(* CoDeSys 2.3.9.50 project: BallGame_template_with_PackMLandDriveFB.pro *)
(* Libraries: TcBase.lib 14.5.09 11:14:08, TcSystem.lib 7.6.16 10:01:22, STANDARD.LIB 5.6.98 11:03:02 *)

(* Task configuration *)
TASK BallGame (PRIORITY := 1, INTERVAL := T#10ms);
	PRG_HMI();
	MAIN();
END_TASK
TASK Drive (PRIORITY := 0, INTERVAL := T#5ms);
	PRG_Drive_Link();
END_TASK

(* Global variable list: Global_Variables *)
VAR_GLOBAL
(* -------------INPUTS and OUTPUTS -------------------*)
(* See Global_Variables_TwinCAT and Global_Variables_CodeSys for
environment specific physical IOs *)

(*-----------------------TIMERS----------------------------*)
	TONMove_Ball_Delay	: TON;
	TONDrive_Delay		: TON;

(*-----------------------COUNTERS----------------------------*)
	CountBallsSortedMetal			: INT:=0;	(*Balls sorted: Metal*)
	CountBallsSortedWooden		: INT:=0;	(*Balls sorted: Wood*)
	CountBallsSortedYellow		: INT:=0;	(*Balls sorted: Wood, Yellow*)
	CountBallsSortedRed			: INT:=0;	(*Balls sorted: Wood, Red*)
	CountBallsSortedBlue			: INT:=0;	(*Balls sorted: Wood, Blue*)
	CountBallsSortedGarbage		: INT:=0;	(*Balls sorted: Unknown*)
	arrCountBallsOnTubes	: ARRAY [1..4] OF INT;	(*Balls on tubes: 1=lower, 2=middle, 3=upper, 4=garbage*)

(*-----------------------FUNCTION BLOCKS----------------*)
	fbDrive				: FB_DriveMovement2;		(*FB for executing the motion*)
	fbStateModel			: FB_StateModel_ST;		(*FB for executing state model*)

(* -------------HMI INPUTS (from HMI to PLC) -------------------*)
	bHMI_BtnStart		: BOOL;		(*Start button on HMI*)
	HMI_uModeReq		: UINT :=1;

(* -------------HMI OUTPUTS (from PLC to HMI) -------------------*)
	PLC_uModeCurrent	: UINT;		(*Current Mode*)
	PLC_uStateCurrent	: UINT;		(*Current State*)
	O_Light_BeaconRed	: BOOL;		(*Light beacon: Red*)

(*-----------------------OTHER GLOBAL VARS ----------------*)


END_VAR

VAR_GLOBAL CONSTANT
(*-----------------------Lift Position Constants----------------------------*)
	GPOS_LOADING		: WORD := 16#0A;	(*Drive to loading level*)
	GPOS_PIPE_LOW	: WORD := 16#0B;	(*Drive to lower pipe*)
	GPOS_PIPE_MID		: WORD := 16#0C;	(*Drive to middle pipe*)
	GPOS_PIPE_UP		: WORD := 16#0D;	(*Drive to upper pipe*)
	GPOS_GARBAGE		: WORD := 16#0E;	(*Drive to garbage pipe*)
	GPOS_COLOR_SEN	: WORD := 16#0F;	(*Drive to colour sensor*)

(*-----------------------Ball Type Constants----------------------------*)
	METAL				: BOOL := FALSE;
	WOODEN		: BOOL := TRUE;

(*-----------------------TIME Constants----------------------------*)
	T_LOADING_BALL	: TIME := T#1.5s;	(*Delay for ball to roll from Slot2 to Lifter*)
	T_DRIVE_DELAY		: TIME := T#2s;	(*Delay for drive to start movement*)
END_VAR

(* Global variable list: Global_Variables_CodeSys *)
VAR_GLOBAL
(* -------------INPUTS-------------------*)
	ISensorOpt 			:BOOL;	(*Optical sensor - is ball present*)
	ISensorInd 			:BOOL;	(*Inductive sensor - is metal ball present*)
	IEmergencyClear 		:BOOL;	(*Emergency stop is cleared*)
	IRun 				:BOOL;	(*Run switch*)
	ILimitUp 				:BOOL;	(*Lift's limit switch is activated - Up*)
	ILimitLow 		 	:BOOL;	(*Lift's limit switch is activated - Low*)
	IGateClosedMid		:BOOL;	(*Pipe gate closed - Mid*)
	IGateClosedLow		:BOOL;	(*Pipe gate closed - Low*)
	ISorterGateClosed		:BOOL;	(*Sorter gate closed*)
	ISorterLiftUp			:BOOL;	(*Sorter lift at up position*)
	ISorterLiftDown		:BOOL;	(*Sorter lift at down position*)
	IPressureApplied		:BOOL;	(*Pressure is available for the system*)
	TEMP1				:BOOL;
	ISenColourYellow		:BOOL;	(*Colour sensor In1 - Yellow*)
	ISenColourBlue		:BOOL;	(*Colour sensor In2 - Blue*)
	ISenColourGreen		:BOOL;	(*Colour sensor In3 - Green*)
	ISenColourRed		:BOOL;	(*Colour sensor In4 - Red*)
	IDriveStatus 			:WORD;	(*From lift drive status information*)

(* -------------OUTPUTS-------------------*)
	OGateMid			:BOOL;	(*Valve: Open pipe gate - Mid*)
	OGateLow			:BOOL;	(*Valve: Open pipe gate - Low*)
	OSorterGate			:BOOL;	(*Valve: Open sorter gate*)
	OSorterLift			:BOOL;	(*Valve: Sorter lift up*)
	OEjector			:BOOL;	(*Ejector push ball out from lift*)
	ODriveControl 		:WORD;	(*To lift drive control information*)
END_VAR

(* Global variable list: Global_Variables_TwinCAT *)
VAR_GLOBAL
(* -------------INPUTS-------------------*)
	ISensorOpt 			AT %I*	:BOOL;	(*Optical sensor - is ball present*)
	ISensorInd 			AT %I*	:BOOL;	(*Inductive sensor - is metal ball present*)
	IEmergencyClear 	AT %I*	:BOOL;	(*Emergency stop is cleared*)
	IRun 				AT %I*	:BOOL;	(*Run switch*)
	ILimitUp 			AT %I*	:BOOL;	(*Lift's limit switch is activated - Up*)
	ILimitLow 			AT %I* 	:BOOL;	(*Lift's limit switch is activated - Low*)
	IGateClosedUp		AT %I* 	:BOOL;
	IGateClosedMid		AT %I*	:BOOL;	(*Pipe gate closed - Mid*)
	IGateClosedLow		AT %I*	:BOOL;	(*Pipe gate closed - Low*)
	ISorterGateClosed	AT %I*	:BOOL;	(*Sorter gate closed*)
	ISorterLiftUp		AT %I*	:BOOL;	(*Sorter lift at up position*)
	ISorterLiftDown		AT %I*	:BOOL;	(*Sorter lift at down position*)
	IPressureApplied	AT %I*	:BOOL;	(*Pressure is available for the system*)
	TEMP1				AT %I*	:BOOL;
	ISenColourYellow	AT %I*	:BOOL;	(*Colour sensor In1 - Yellow*)
	ISenColourBlue		AT %I*	:BOOL;	(*Colour sensor In2 - Blue*)
	ISenColourGreen		AT %I*	:BOOL;	(*Colour sensor In3 - Green*)
	ISenColourRed		AT %I*	:BOOL;	(*Colour sensor In4 - Red*)
	IDriveStatus 		AT %I*	:WORD;	(*From lift drive status information*)

(* -------------OUTPUTS-------------------*)
	OGateUp				AT %Q*	:BOOL;
	OGateMid			AT %Q*	:BOOL;	(*Valve: Open pipe gate - Mid*)
	OGateLow			AT %Q*	:BOOL;	(*Valve: Open pipe gate - Low*)
	OSorterGate			AT %Q*	:BOOL;	(*Valve: Open sorter gate*)
	OSorterLift			AT %Q*	:BOOL;	(*Valve: Sorter lift up*)
	OEjector			AT %Q*	:BOOL;	(*Ejector push ball out from lift*)
	ODriveControl 		AT %Q*	:WORD;	(*To lift drive control information*)

(* -------------HMI-------------------*)
	I_Btn_Reset		: BOOL;	(*Button: Reset*)
	I_Btn_Start		: BOOL;	(*Button: Start*)
	I_Btn_Stop		: BOOL;	(*Button: Stop*)
	I_Btn_EStop		: BOOL;	(*Button: Reset*)

(* -------------Drive-------------------*)
	bDriveEnabled 	: BOOL;

END_VAR

(* Global variable list: TwinCAT_Configuration *)
(* Generated automatically by TwinCAT - (read only) *)
VAR_CONFIG
	.ISensorOpt AT %IX0.0 : BOOL;	(*  ~ {LinkedWith:TIID^Device 4 (EL6731)^Box 2  (BK3110)^Term 2 (KL1002)^Channel 1^Input} *)
	.ISensorInd AT %IX0.1 : BOOL;	(*  ~ {LinkedWith:TIID^Device 4 (EL6731)^Box 2  (BK3110)^Term 2 (KL1002)^Channel 2^Input} *)
	.IEmergencyClear AT %IX0.2 : BOOL;	(*  ~ {LinkedWith:TIID^Device 4 (EL6731)^Box 2  (BK3110)^Term 3 (KL1002)^Channel 1^Input} *)
	.IRun AT %IX0.3 : BOOL;	(*  ~ {LinkedWith:TIID^Device 4 (EL6731)^Box 2  (BK3110)^Term 3 (KL1002)^Channel 2^Input} *)
	.ILimitUp AT %IX0.4 : BOOL;	(*  ~ {LinkedWith:TIID^Device 4 (EL6731)^Box 2  (BK3110)^Term 4 (KL1002)^Channel 1^Input} *)
	.ILimitLow AT %IX0.5 : BOOL;	(*  ~ {LinkedWith:TIID^Device 4 (EL6731)^Box 2  (BK3110)^Term 4 (KL1002)^Channel 2^Input} *)
	.IGateClosedUp AT %IX8.0 : BOOL;
	.IGateClosedMid AT %IX0.7 : BOOL;	(*  ~ {LinkedWith:TIID^Device 4 (EL6731)^Box 2  (BK3110)^Term 5 (KL1104)^Channel 2^Input} *)
	.IGateClosedLow AT %IX1.0 : BOOL;	(*  ~ {LinkedWith:TIID^Device 4 (EL6731)^Box 2  (BK3110)^Term 5 (KL1104)^Channel 3^Input} *)
	.ISorterGateClosed AT %IX1.1 : BOOL;	(*  ~ {LinkedWith:TIID^Device 4 (EL6731)^Box 2  (BK3110)^Term 5 (KL1104)^Channel 4^Input} *)
	.ISorterLiftUp AT %IX1.2 : BOOL;	(*  ~ {LinkedWith:TIID^Device 4 (EL6731)^Box 2  (BK3110)^Term 6 (KL1104)^Channel 1^Input} *)
	.ISorterLiftDown AT %IX1.3 : BOOL;	(*  ~ {LinkedWith:TIID^Device 4 (EL6731)^Box 2  (BK3110)^Term 6 (KL1104)^Channel 2^Input} *)
	.IPressureApplied AT %IX1.4 : BOOL;	(*  ~ {LinkedWith:TIID^Device 4 (EL6731)^Box 2  (BK3110)^Term 6 (KL1104)^Channel 3^Input} *)
	.TEMP1 AT %IX1.5 : BOOL;	(*  ~ {LinkedWith:TIID^Device 4 (EL6731)^Box 2  (BK3110)^Term 6 (KL1104)^Channel 4^Input} *)
	.ISenColourYellow AT %IX1.6 : BOOL;	(*  ~ {LinkedWith:TIID^Device 4 (EL6731)^Box 2  (BK3110)^Term 7 (KL1104)^Channel 1^Input} *)
	.ISenColourBlue AT %IX1.7 : BOOL;	(*  ~ {LinkedWith:TIID^Device 4 (EL6731)^Box 2  (BK3110)^Term 7 (KL1104)^Channel 2^Input} *)
	.ISenColourGreen AT %IX2.0 : BOOL;	(*  ~ {LinkedWith:TIID^Device 4 (EL6731)^Box 2  (BK3110)^Term 7 (KL1104)^Channel 3^Input} *)
	.ISenColourRed AT %IX2.1 : BOOL;	(*  ~ {LinkedWith:TIID^Device 4 (EL6731)^Box 2  (BK3110)^Term 7 (KL1104)^Channel 4^Input} *)
	.IDriveStatus AT %IB4 : WORD;	(*  ~ {LinkedWith:TIID^Device 4 (EL6731)^Box 5 (DKC03)^DKC03 mit LSPM2^Inputs^DKC03 mit LSPM2_0_0} *)
	.OGateUp AT %QX4.0 : BOOL;
	.OGateMid AT %QX0.1 : BOOL;	(*  ~ {LinkedWith:TIID^Device 4 (EL6731)^Box 2  (BK3110)^Term 8 (KL2114)^Channel 2^Output} *)
	.OGateLow AT %QX0.2 : BOOL;	(*  ~ {LinkedWith:TIID^Device 4 (EL6731)^Box 2  (BK3110)^Term 8 (KL2114)^Channel 3^Output} *)
	.OSorterGate AT %QX0.3 : BOOL;	(*  ~ {LinkedWith:TIID^Device 4 (EL6731)^Box 2  (BK3110)^Term 8 (KL2114)^Channel 4^Output} *)
	.OSorterLift AT %QX0.4 : BOOL;	(*  ~ {LinkedWith:TIID^Device 4 (EL6731)^Box 2  (BK3110)^Term 9 (KL2114)^Channel 1^Output} *)
	.OEjector AT %QX0.5 : BOOL;	(*  ~ {LinkedWith:TIID^Device 4 (EL6731)^Box 2  (BK3110)^Term 9 (KL2114)^Channel 2^Output} *)
	.ODriveControl AT %QB2 : WORD;	(*  ~ {LinkedWith:TIID^Device 4 (EL6731)^Box 5 (DKC03)^DKC03 mit LSPM2^Outputs^DKC03 mit LSPM2_1_0} *)
END_VAR

(* Data type *)
TYPE E_BallColour :
(
	NoColour := 0,
	Yellow := 1,
	Blue := 2,
	Red := 3
);
END_TYPE

(* Data type *)
TYPE E_ModeCtrl :
(
	eMode_undefined := 0,
	eMode_Automatic :=1,
	eMode_XXX :=2,
	eMode_Manual :=99
);
END_TYPE

(* Data type *)
TYPE E_ModeProc :
(*Procedural control modes. Can be changed in any state*)
(
	eModeProc_undefined := 0,
	eModeProc_Automatic :=1,
	eModeProc_SemiAutomatic :=2,
	eModeProc_Manual :=3
);
END_TYPE

(* Data type *)
TYPE E_State :
(
	eSt_Aborting :=0,
	eSt_Aborted,
	eSt_Clearing,
	eSt_Stopped,
	eSt_Stopping,
	eSt_Resetting,
	eSt_Idle,
	eSt_Starting,
	eSt_Execute,
	eSt_Suspending,
	eSt_Suspended,
	eSt_Unsuspending,
	eSt_Holding,
	eSt_Held,
	eSt_UnHolding,
	eSt_Completing,
	eSt_Completed
);
END_TYPE

(* POU PRG_HMI, ST *)
PROGRAM PRG_HMI
VAR
	(*HMI Buttons*)
	bBtnResetCounters	: BOOL;	(*Button Reset counters*)
	bBtnEmptyPipes		: BOOL;	(*Button Empty Pipes*)

	(*Variables for Lift visualisation*)
	iSorterLiftPos	: INT;		(*Position of Sorter Lift cylinder*)
	iLiftPos		: INT;		(*Position of the lift*)
	wTargetPos	: INT;		(*Current target position of the lift*)
	bBall_InLift	: BOOL;		(*Is there a ball in lift*)

	(*internal variables*)
	RS_Ball_InLift	: RS;		(*Flip-flop for ball in the lift*)
	i: INT := 0;		(*Counter*)
END_VAR
(*Producing blinking signal*)
PRG_Blinking();

(*Sorter lift position calculus*)
IF OSorterLift AND (iSorterLiftPos < 30) THEN
	iSorterLiftPos := iSorterLiftPos +1;
END_IF;
IF NOT OSorterLift AND (iSorterLiftPos > 0) THEN
	iSorterLiftPos := iSorterLiftPos - 1;
END_IF;

(*Lift position calculus*)
CASE fbDrive.wDestination OF
GPOS_PIPE_UP:		(*Go to Pipe Up*)
	wTargetPos:=375;
GPOS_PIPE_MID:	(*Go to Pipe Mid*)
	wTargetPos:=275;
GPOS_COLOR_SEN:	(*Go to Colour sensor*)
	wTargetPos:=220;
GPOS_PIPE_LOW:	(*Go to Pipe Low*)
	wTargetPos:=175;
GPOS_GARBAGE:	(*Go to garbage position*)
	wTargetPos:=110;
GPOS_LOADING:	(*Go to loading position*)
	wTargetPos:=20;
ELSE
	wTargetPos:=0;
END_CASE;

(*Drive lift*)
IF iLiftPos > wTargetPos THEN	(*Lift is higher than target*)
	iLiftPos := iLiftPos - 1;	 (*Go down*)
ELSIF iLiftPos < wTargetPos THEN	(*Lift is lower than target*)
	iLiftPos := iLiftPos + 1;	 (*Go up*)
END_IF;

(*Is there a ball in the lift*)
RS_Ball_InLift(
	SET:= (iLiftPos=20 AND NOT OSorterGate),
	RESET1:=OEjector ,
	Q1=>bBall_InLift );

(* ---------------------------------- Button handlers ---------------------------------- *)
(*Button Empty Pipes*)

(*Button Reset coutners*)
IF bBtnResetCounters THEN
	CountBallsSortedMetal := 0;
	CountBallsSortedWooden := 0;
	CountBallsSortedYellow := 0;
	CountBallsSortedBlue := 0;
	FOR i := 1 TO 3 DO
		arrCountBallsOnTubes[i] := 0;
	END_FOR;
END_IF;
END_PROGRAM

(* POU Programs/PRG_Blinking, ST *)
PROGRAM PRG_Blinking
(*Supporting caluculations: Blinking signals
Author: 	Niko Siltala, niko.siltala@tut.fi
Date: 	2014-01-01*)

VAR_OUTPUT
	bSign4Hz	:BOOL;				(*4 Hz (240krt/min) taajudella vaihteleva signaali*)
	bSign2Hz	:BOOL;				(*2 Hz (120krt/min) taajudella vaihteleva signaali*)
	bSign1Hz	:BOOL;				(*1 Hz (60krt/min) taajudella vaihteleva signaali*)
	bSign0_5Hz	:BOOL;				(*0,5 Hz (30krt/min) taajudella vaihteleva signaali*)
END_VAR
VAR
	bInitDone	: BOOL	:=FALSE;		(*Ohjelman initialisointi*)
	TP_Delay	: TP;					(*Nopein taajuus / 2 tuottaja*)
	bBaseHz	: BOOL	:=FALSE;		(*Nopein taajuus/2*)
	iBaseHz		: UINT	:=4;			(*Base taajuus (Hz)*)
	RTRIG_2Hz_Sign 	: R_TRIG;		(*2Hz signaalin generointi*)
	RTRIG_1Hz_Sign 	: R_TRIG;		(*1Hz signaalin generointi*)
	RTRIG_0_5Hz_Sign	: R_TRIG;	(*0,5Hz signaalin generointi*)
	tBaseTaajuus	:TIME;			(*Base vilkutuksen timerin arvo. f/2*)
	fPLC_CYCLE_TIME	: LREAL;		(*PLC:n cycli aika. Sekunttia*)
END_VAR
(*Ohjelman initialisoinnit - Suoritetaan vain kertaalleen*)
IF NOT bInitDone THEN
	fPLC_CYCLE_TIME := UDINT_TO_LREAL(SystemTaskInfoArr[1].cycleTime) / 10E6;
	(*Base Vilkkusignaalien tuottaminen*)
	(* 250ms - 1* cykliaika(20ms)*)
	tBaseTaajuus := LREAL_TO_TIME( ( (1/ UINT_TO_LREAL(iBaseHz) / 2 ) - 1 * fPLC_CYCLE_TIME ) * 1000);
	bInitDone := TRUE;
END_IF;


(*Base signaalin genrointi*)
TP_Delay(IN:=NOT TP_Delay.Q , PT:=tBaseTaajuus);
IF NOT TP_Delay.Q THEN
	bBaseHz := NOT bBaseHz;
	bSign4Hz:= bBaseHz;
END_IF;

(*2Hz signaalin genrointi*)
RTRIG_2Hz_Sign(CLK:=bSign4Hz);
IF RTRIG_2Hz_Sign.Q THEN
	bSign2Hz:=NOT bSign2Hz;
END_IF;

(*1Hz signaalin genrointi*)
RTRIG_1Hz_Sign(CLK:=bSign2Hz);
IF RTRIG_1Hz_Sign.Q THEN
	bSign1Hz:=NOT bSign1Hz;
END_IF;

(*0,5 Hz signaalin generointi*)
RTRIG_0_5Hz_Sign(CLK:=bSign1Hz);
IF (RTRIG_0_5Hz_Sign.Q) THEN
	bSign0_5Hz:= NOT bSign0_5Hz;
END_IF;
END_PROGRAM

(* POU MAIN, ST *)
PROGRAM MAIN
(*Main program for application. Uses PackML state model to control the execution of the application*)
VAR
	tonStarting			: TON;
	rsEmergencyClear	: RS;	(*RS - flip-flop for Emergency clear info*)
END_VAR
(* ****** Section 1: Initialisations and default values. Initial conditions for variables on every PLC cycle*)
(*Default values*)
fbStateModel.bSC := FALSE;
(*System resets*)

(* ****** Section 2: Actions in your program without considering the Control Mode. I.e. actions are performed same way indenpendent on
current Control Mode selection.*)
(*Mode independent state actions. Change / Add / Remove states according your need*)
CASE fbStateModel.eState OF
eSt_Aborting:
	(* One can make specific actions in case of specific Mode-State combination.
	   One can also consider to call a specific program when in specific Mode-State combination*)
	actAborting;
	fbStateModel.bSC := TRUE;		(*MODIFY*)
eSt_Clearing:
	fbStateModel.bSC := TRUE;		(*MODIFY*)
eSt_Resetting:
	fbStateModel.bSC := TRUE;
eSt_Holding:
	fbStateModel.bSC := TRUE;		(*MODIFY*)
eSt_UnHolding:
	fbStateModel.bSC := TRUE;		(*MODIFY*)
eSt_Suspending:
	fbStateModel.bSC := TRUE;		(*MODIFY*)
eSt_Unsuspending:
	fbStateModel.bSC := TRUE;		(*MODIFY*)
END_CASE;

(* ****** Section 3: Actions in your program which are Control Mode specific. Two nested case structures where outer one selects the
control mode and inner the PackML state. In order to avoid conflicts, it would be better to process each PackML state either in Section 2 
or Section 3, but not in both. *)
(*Execution mode related state actions. Change / Add / Remove mode and states according your need*)
CASE fbStateModel.eMode OF
(*MODE: MANUAL*)
eMode_Manual:
	(* ****** Section 3.1: PackML state based processing actions when Control Mode is Manual.*)
	CASE fbStateModel.eState OF
	eSt_Starting:
		IF IPressureApplied THEN
			fbStateModel.bSC := TRUE;			(*MODIFY*)
		END_IF
	eSt_Stopping:
		fbStateModel.bSC := TRUE;			(*MODIFY*)
	END_CASE;

(*MODE: AUTOMATIC*)
eMode_Automatic:
	(* ****** Section 3.2: PackML state based processing actions when Control Mode is Automatic.*)
	CASE fbStateModel.eState OF
	eSt_Idle:
		tonStarting(IN:=FALSE , PT:= , Q=> , ET=> );	(*MODIFY*)
	eSt_Starting:
		(* tonStarting(IN:=TRUE , PT:=T#2s , Q=> , ET=> );
		fbStateModel.bSC := tonStarting.Q; *)
		IF IPressureApplied THEN
			bDriveEnabled := TRUE;
			PRG_Initialisation(bReset:= , bExecute:= TRUE , bDone=> );
		END_IF

		IF PRG_Initialisation.bDone THEN
			PRG_Initialisation(bReset:= , bExecute:= FALSE , bDone=> );
			fbStateModel.bSC := TRUE;
		END_IF
	eSt_Completing:
		fbStateModel.bSC := TRUE;					(*MODIFY*)
	eSt_Completed:
		;
	END_CASE;

(* ****** Section 4: Grouping PackML states for calling Programs or FB instances.
This is to avoid repetition inside above case structure in Section 3. With IF clause setting lower (and upper) state limits we can filter out the states when we want to call 
specific programs. The order of states is defined in Tab:Data types > E_PackMLState. eSt_Aborting is lowest and eSt_Completed is highest.
Here we filter calling programs, only when we are in higher states than Stopped. 
This can be pulled out as completely separated section, like in PackML_StateModel_v2-2.pro project. There is inside IF again CASE which process each Control Mode separately.*)
(*Execution part. Making calls for program if we are on states above Stopped*)
	(*If we are between specific states, make some action or program call*)
	IF  (fbStateModel.eState>eSt_Starting) AND (fbStateModel.eState<=eSt_Completing) THEN
		(*Make here the actions / calls Good place to start with is PRG_Sorting (PRG)*)
		PRG_AutoSort(bExecute:= TRUE , bReset:= , bDone=> , bStopOk=> );
	END_IF;

(*MODE: UNKNOWN*)
ELSE	(*Error*)
	; (*TODO*)
END_CASE;

(* ****** Section 5: Calling the fbStateModel instance.
Here the instance of state model is called and all triggering inputs are set, but bSC (State Completed), which you control in your programs. 
This is indication that your program has  finished certain stage.
- Pay attention where the instance fbStateModel is defined. Do you do it in global variables or e.g. here in PRG_MAIN? Important is to use the 
same instance in all places, so that machine state is unique and shared. Remember, if you have multiple definitions, the PRG_MAIN "hides" 
the global one, and might lead to problems elswhere, when you think you are using the same instance, but actually are not. 
- In case you are using the PackML visualisation (VC_PackMLStates), make sure you connect its placeholder to the very same PackML FB instance.
- The Mask for wIgnoreState is created as following. I use binary base for the value(2#). The lowest bit in the mask corresponds the eSt_Aborting
 in E_PackMLState. The next is eSt_Aborted, and so on. Specific state is ignored and jumped over when it is masked out i.e. ignored by having 1 
in that position. Note that implementation allows this only for selected states. See FB_PackMLStateModel_ST code for further details.*)
(*Calling & Updating the state model*)
(*TODO: Evaluate and change all input conditions according your application needs*)
fbStateModel(
	bResetFB:= ,
	eModeReq:= HMI_uModeReq,
	wIgnoreState := 2#000000,		(*TODO: Which states should be ignodered. Default: 2#000000 or 2#100000. The latter is ignoring Resetting state*)
	bSC:= ,			(*Must not be assigned ANY variable, because fb input is directly operated!!!*)
	bAbort:= NOT (IEmergencyClear  OR  IPressureApplied),
	bClear:= IEmergencyClear,
	bReset:= I_Btn_Start,
	bStart:= I_Btn_Start,
	bHold:= ,
	bUn_Hold:= ,
	bSuspend:= ,
	bUn_Suspend:= ,
	bStop:= I_Btn_Stop ,
	bComplete:= ,
	bAck_Completed:= ,
	eMode=> PLC_uModeCurrent,
	eState=> PLC_uStateCurrent);

(* ****** Section 6: Here we update all outputs according the current state of our PackML model. This allows us to process the in single location.
The control of outputs is bind to state, not e.g. to inputs. The inputs are the one driving the PackML model forward. Again CASE structure can be used.*)
(*Call for HMI and UI update*)
(*PRG_Drive_Link()*);
HMI_and_UI_Update;
END_PROGRAM
ACTION actAborting:
bDriveEnabled := FALSE;
PRG_Sorting(bReset:=TRUE , bExecute:= FALSE);
END_ACTION
ACTION HMI_and_UI_Update:
(*Simulate emergency stop circuitry
rsEmergencyClear(
	SET:= I_Btn_Reset,
	RESET1:= I_Btn_EStop ,
	Q1=> IEmergencyClear);
*)

(*HMI Update*)
PRG_Blinking (bSign4Hz=> , bSign2Hz=> , bSign1Hz=> , bSign0_5Hz=> );
(*Init values*)
O_Light_BeaconRed := FALSE;

(*OLight_Start :=  (fbStateModel.eState >= eSt_Resetting) AND (fbStateModel.eState < eSt_Completed);*)
CASE fbStateModel.eState OF
eSt_Aborting, eSt_Aborted:
	O_Light_BeaconRed := PRG_Blinking.bSign1Hz;
eSt_Clearing:
	O_Light_BeaconRed := PRG_Blinking.bSign0_5Hz;
eSt_Stopped, eSt_Completed:
	O_Light_BeaconRed := TRUE;
eSt_Starting:
	;
END_CASE;
END_ACTION

(* POU Programs/PRG_Initialisation, SFC *)
PROGRAM PRG_Initialisation
(*Template program for system initialisation*)
VAR_INPUT
	bReset	: BOOL := FALSE;	(*Reseting the SFC*)
	bExecute	: BOOL;			(*Executes PRG*)
END_VAR
VAR_OUTPUT
	bDone		: BOOL;		(*Program operations done*)
END_VAR
VAR
(* -------------INTERNAL-------------------*)
	tonMoveDelay		: TON;
	tMoveDelay		: TIME := T#1s;
	bInitDone			: BOOL:=FALSE;	(*Initialisation done*)
	bGatesClosed	: BOOL:=FALSE;	(*Initialisation done*)
	bActuRetracted	: BOOL:=FALSE;
	bDriveAtLoading	: BOOL:=FALSE;

(*System variables. See SFC-flags: http://infosys.beckhoff.com/content/1033/tcplccontrol/html/tcplcctrl_editorsfc.htm?id=24319#SFC-Flags*)
	SFCReset		: BOOL := FALSE;	(*For reseting the SFC*)
END_VAR
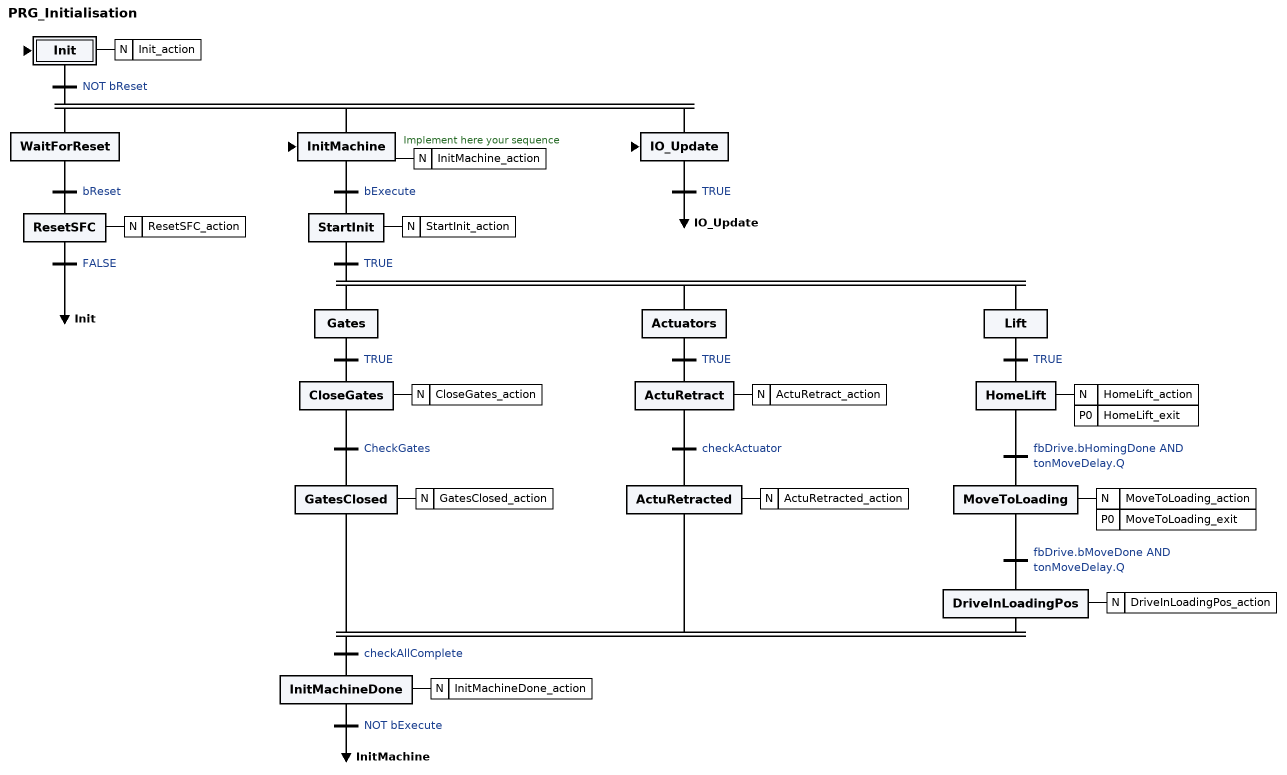
INITIAL_STEP Init:
	Init_action(N);
END_STEP
TRANSITION FROM Init TO (WaitForReset, InitMachine, IO_Update) := NOT bReset;
END_TRANSITION
STEP WaitForReset:
END_STEP
TRANSITION FROM WaitForReset TO ResetSFC := bReset;
END_TRANSITION
STEP InitMachine: (* Implement here your sequence *)
	InitMachine_action(N);
END_STEP
TRANSITION FROM InitMachine TO StartInit := bExecute;
END_TRANSITION
STEP StartInit:
	StartInit_action(N);
END_STEP
TRANSITION FROM StartInit TO (Gates, Actuators, Lift) := TRUE;
END_TRANSITION
STEP Gates:
END_STEP
TRANSITION FROM Gates TO CloseGates := TRUE;
END_TRANSITION
STEP CloseGates:
	CloseGates_action(N);
END_STEP
TRANSITION FROM CloseGates TO GatesClosed := CheckGates;
END_TRANSITION
STEP GatesClosed:
	GatesClosed_action(N);
END_STEP
STEP Actuators:
END_STEP
TRANSITION FROM Actuators TO ActuRetract := TRUE;
END_TRANSITION
STEP ActuRetract:
	ActuRetract_action(N);
END_STEP
TRANSITION FROM ActuRetract TO ActuRetracted := checkActuator;
END_TRANSITION
STEP ActuRetracted:
	ActuRetracted_action(N);
END_STEP
STEP Lift:
END_STEP
TRANSITION FROM Lift TO HomeLift := TRUE;
END_TRANSITION
STEP HomeLift:
	HomeLift_action(N);
	HomeLift_exit(P0);
END_STEP
TRANSITION FROM HomeLift TO MoveToLoading := fbDrive.bHomingDone AND tonMoveDelay.Q;
END_TRANSITION
STEP MoveToLoading:
	MoveToLoading_action(N);
	MoveToLoading_exit(P0);
END_STEP
TRANSITION FROM MoveToLoading TO DriveInLoadingPos := fbDrive.bMoveDone AND tonMoveDelay.Q;
END_TRANSITION
STEP DriveInLoadingPos:
	DriveInLoadingPos_action(N);
END_STEP
TRANSITION FROM (GatesClosed, ActuRetracted, DriveInLoadingPos) TO InitMachineDone := checkAllComplete;
END_TRANSITION
STEP InitMachineDone:
	InitMachineDone_action(N);
END_STEP
TRANSITION FROM InitMachineDone TO InitMachine := NOT bExecute;
END_TRANSITION
STEP IO_Update:
END_STEP
TRANSITION FROM IO_Update TO IO_Update := TRUE;
END_TRANSITION
STEP ResetSFC:
	ResetSFC_action(N);
END_STEP
TRANSITION FROM ResetSFC TO Init := FALSE;
END_TRANSITION

ACTION Init_action:
(*Clear Reset SFC*)
SFCReset:= FALSE;
bDone := FALSE;
END_ACTION

ACTION InitMachine_action:
(*Do some actions...

Sulje kaikki portit ... JA tarkista Steppiä seuraavassa transitioehdossa, että kaikki portit ovat kiinni
Close all gates.... and check in following transition that ALL gates are closed*)

;
END_ACTION

ACTION StartInit_action:
bDone := FALSE;
END_ACTION

ACTION CloseGates_action:
OGateUp		:= FALSE;
OGateMid	:= FALSE;
OGateLow	:= FALSE;
OSorterGate	:= FALSE;
END_ACTION

ACTION GatesClosed_action:
bGatesClosed := TRUE;
END_ACTION

ACTION ActuRetract_action:
OSorterLift	 := FALSE;
OEjector	 := FALSE;
END_ACTION

ACTION ActuRetracted_action:
bActuRetracted := TRUE;
END_ACTION

ACTION HomeLift_action:
fbDrive.bEnable := TRUE;
fbDrive.bStart := TRUE;
tonMoveDelay(IN:=TRUE , PT:= tMoveDelay);
END_ACTION

ACTION HomeLift_exit:
fbDrive.bStart:= FALSE;
tonMoveDelay(IN:=FALSE);
END_ACTION

ACTION MoveToLoading_action:
fbDrive.wTarget := GPOS_LOADING;
fbDrive.bStart:= TRUE;
tonMoveDelay(IN:=TRUE , PT:= tMoveDelay);
END_ACTION

ACTION MoveToLoading_exit:
fbDrive.bStart:= FALSE;
tonMoveDelay(IN:=FALSE);
END_ACTION

ACTION DriveInLoadingPos_action:
bDriveAtLoading := TRUE;
END_ACTION

ACTION InitMachineDone_action:
bDone := TRUE;
END_ACTION

ACTION ResetSFC_action:
(*Reset SFC*)
SFCReset:=TRUE;
END_ACTION

TRANSITION CheckGates:
_FBD_ (* Function Block Diagram *)
NETWORK 1
	AND(IGateClosedUp, IGateClosedMid, IGateClosedLow, ISorterGateClosed)
_END_FBD_
END_TRANSITION

TRANSITION checkActuator:
_FBD_ (* Function Block Diagram *)
NETWORK 1
	AND(ISorterLiftDown, NOT OEjector)
_END_FBD_
END_TRANSITION

TRANSITION checkAllComplete:
_FBD_ (* Function Block Diagram *)
NETWORK 1
	AND(bGatesClosed, bActuRetracted, bDriveAtLoading)
_END_FBD_
END_TRANSITION
END_PROGRAM

(* POU Programs/PRG_AutoSort, ST *)
PROGRAM PRG_AutoSort
VAR_INPUT
	bExecute	: BOOL;
	bReset	: BOOL := FALSE;
END_VAR
VAR_OUTPUT
	bDone		: BOOL;		(*Program operations done*)
	bStopOk    : BOOL;
END_VAR
VAR
	fbSorter	: FB_Sorter;
	fbLift		: FB_Lift;
	bBatchComplete  : BOOL := FALSE;
END_VAR
actUpdateIO;
actCheckAllOkStop;

CASE fbStateModel.eState OF
	eSt_Idle:
		fbStateModel.bComplete  := FALSE;
		fbStateModel.bSC 		:= TRUE;
	eSt_Resetting:
		fbStateModel.bSC := TRUE;
	eSt_Stopping:
		fbStateModel.bStop := FALSE;

		IF  bStopOk THEN
			fbStateModel.bSC := TRUE;
		END_IF
	eSt_Execute:
		fbSorter (bEnable :=  TRUE , bReset := FALSE);
		fbLift(bEnable :=  TRUE , bReset := FALSE);
		IF bBatchComplete  THEN
			fbStateModel.bComplete := TRUE;
		END_IF

	eSt_Completing:
		fbStateModel.bComplete := FALSE;
		IF bStopOK THEN
			fbStateModel.bSC := TRUE;
		END_IF

	eSt_Unsuspending:
		fbStateModel.bSC := TRUE;

	eSt_Suspending:
		fbStateModel.bSuspend := FALSE;
		fbStateModel.bSC := TRUE;

END_CASE
END_PROGRAM
ACTION actCheckAllOKStop:
IF fbSorter.bStopOK AND  fbLift.bStopOK THEN
	bStopOK := TRUE;
ELSE
	bStopOK := FALSE;
END_IF
END_ACTION
ACTION actUpdateIO:
fbSorter (
	bReset:= ,
	bEnable:= bExecute,
	I_SensorOpt:= ISensorOpt ,
	I_SensorInd:= ISensorInd,
	I_SorterLiftUp:= ISorterLiftUp ,
	I_SorterLiftDown:= ISorterLiftDown,
	hiRdyToReceive_FromDS:= fbLift.hoReadyToRecieve_ToUS ,
	hiBallAvail_FromUS:= ,
	bStopOK=> ,
	bBallLoaded=> ,
	bCurBallMetal=> ,
	O_SorterGate=> OSorterGate ,
	O_SorterLift=> OSorterLift ,
	hoBallAvail_ToDS=> ,
	hoReadyToRecieve_ToUS=> );

fbLift (
	bReset:= ,
	bEnable:= bExecute,
	I_LimitUp:= ILimitUp  ,
	I_LimitLow:= ILimitLow,
	I_WaitingBallMetal:= fbSorter.bCurBallMetal  ,
	I_SenColourYellow:= ISenColourYellow ,
	I_SenColourBlue:= ISenColourBlue ,
	I_SenColourGreen:= ISenColourGreen,
	I_SenColourRed:= ISenColourRed ,
	hiRdyToReceive_FromDS:= ,
	hiBallAvail_FromUS:= fbSorter.hoBallAvail_ToDS ,
	bStopOK=> ,
	bBallLoaded=> , 
	bCurBallMetal=> , 
	O_Ejector=> OEjector ,
	hoBallAvail_ToDS=> , 
	hoReadyToRecieve_ToUS=> );
END_ACTION

(* POU FBs/FB_Sorter, SFC *)
FUNCTION_BLOCK FB_Sorter
VAR_INPUT
	bReset			: BOOL;	(*Reset Request*)
	bEnable			: BOOL;
	I_SensorOpt		: BOOL;
	I_SensorInd		: BOOL;
	I_SorterLiftUp		: BOOL;
	I_SorterLiftDown	: BOOL;

	(*SMEMA Handshake Inputs*)
	hiRdyToReceive_FromDS	: BOOL;
	hiBallAvail_FromUS			: BOOL;
END_VAR
VAR_OUTPUT
	bStopOK			: BOOL;
	bBallLoaded		: BOOL;
	bCurBallMetal		: BOOL;
	O_SorterGate		: BOOL;
	O_SorterLift		: BOOL;

	(*SMEMA Handshake Outputs*)
	hoBallAvail_ToDS				: BOOL;
	hoReadyToRecieve_ToUS	: BOOL;
END_VAR
VAR
	tTransferDelay: TIME := T#2s;
	tMoveDelay	: TIME := T#1s;
	fbDelay		: FB_Wait;
	bLocalReset	: BOOL;	(*Performs local reset*)
	SFCReset 	: BOOL;	(*Resets the execution of SFC to init once this SFCFlag is set true *)
END_VAR
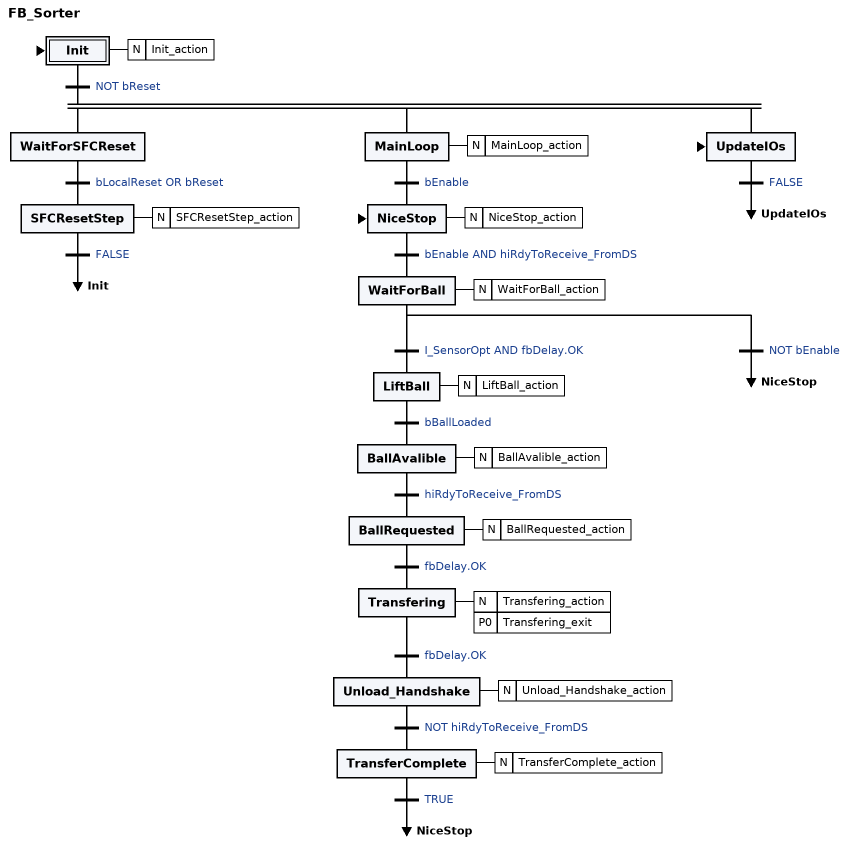
INITIAL_STEP Init:
	Init_action(N);
END_STEP
TRANSITION FROM Init TO (WaitForSFCReset, MainLoop, UpdateIOs) := NOT bReset;
END_TRANSITION
STEP WaitForSFCReset:
END_STEP
TRANSITION FROM WaitForSFCReset TO SFCResetStep := bLocalReset OR bReset;
END_TRANSITION
STEP MainLoop:
	MainLoop_action(N);
END_STEP
TRANSITION FROM MainLoop TO NiceStop := bEnable;
END_TRANSITION
STEP NiceStop:
	NiceStop_action(N);
END_STEP
TRANSITION FROM NiceStop TO WaitForBall := bEnable AND hiRdyToReceive_FromDS;
END_TRANSITION
STEP WaitForBall:
	WaitForBall_action(N);
END_STEP
TRANSITION FROM WaitForBall TO LiftBall := I_SensorOpt AND fbDelay.OK;
END_TRANSITION
TRANSITION FROM WaitForBall TO NiceStop := NOT bEnable;
END_TRANSITION
STEP LiftBall:
	LiftBall_action(N);
END_STEP
TRANSITION FROM LiftBall TO BallAvalible := bBallLoaded;
END_TRANSITION
STEP BallAvalible:
	BallAvalible_action(N);
END_STEP
TRANSITION FROM BallAvalible TO BallRequested := hiRdyToReceive_FromDS;
END_TRANSITION
STEP BallRequested:
	BallRequested_action(N);
END_STEP
TRANSITION FROM BallRequested TO Transfering := fbDelay.OK;
END_TRANSITION
STEP Transfering:
	Transfering_action(N);
	Transfering_exit(P0);
END_STEP
TRANSITION FROM Transfering TO Unload_Handshake := fbDelay.OK;
END_TRANSITION
STEP Unload_Handshake:
	Unload_Handshake_action(N);
END_STEP
TRANSITION FROM Unload_Handshake TO TransferComplete := NOT hiRdyToReceive_FromDS;
END_TRANSITION
STEP TransferComplete:
	TransferComplete_action(N);
END_STEP
TRANSITION FROM TransferComplete TO NiceStop := TRUE;
END_TRANSITION
STEP UpdateIOs:
END_STEP
TRANSITION FROM UpdateIOs TO UpdateIOs := FALSE;
END_TRANSITION
STEP SFCResetStep:
	SFCResetStep_action(N);
END_STEP
TRANSITION FROM SFCResetStep TO Init := FALSE;
END_TRANSITION

ACTION Init_action:
SFCReset := FALSE;
bLocalReset	:= FALSE;
bStopOK := FALSE;
END_ACTION

ACTION MainLoop_action:
hoBallAvail_ToDS			  := FALSE;
hoReadyToRecieve_ToUS := FALSE;
END_ACTION

ACTION NiceStop_action:
bBallLoaded 				  := FALSE;
bStopOK					  := TRUE;
hoBallAvail_ToDS			  := FALSE;
hoReadyToRecieve_ToUS := FALSE;
END_ACTION

ACTION WaitForBall_action:
fbDelay(IN_TIME:=tMoveDelay);
(* Move Lift Down *)
O_SorterLift := FALSE;
END_ACTION

ACTION LiftBall_action:
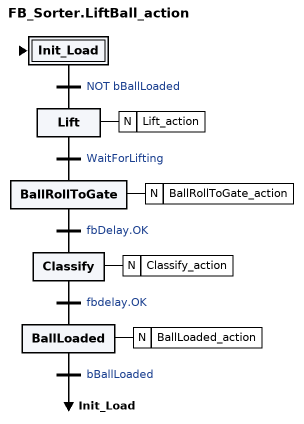
INITIAL_STEP Init_Load:
END_STEP
TRANSITION FROM Init_Load TO Lift := NOT bBallLoaded;
END_TRANSITION
STEP Lift:
	Lift_action(N);
END_STEP
TRANSITION FROM Lift TO BallRollToGate := WaitForLifting;
END_TRANSITION
STEP BallRollToGate:
	BallRollToGate_action(N);
END_STEP
TRANSITION FROM BallRollToGate TO Classify := fbDelay.OK;
END_TRANSITION
STEP Classify:
	Classify_action(N);
END_STEP
TRANSITION FROM Classify TO BallLoaded := fbdelay.OK;
END_TRANSITION
STEP BallLoaded:
	BallLoaded_action(N);
END_STEP
TRANSITION FROM BallLoaded TO Init_Load := bBallLoaded;
END_TRANSITION

ACTION Lift_action:
O_SorterLift := TRUE;
fbDelay(IN_TIME:=tMoveDelay);
END_ACTION

ACTION BallRollToGate_action:
fbDelay(IN_TIME:=tMoveDelay);
END_ACTION

ACTION Classify_action:
fbDelay(IN_TIME:=tMoveDelay);
IF I_SensorInd THEN
	bCurBallMetal := FALSE;
ELSE
	bCurBallMetal := TRUE;
END_IF
END_ACTION

ACTION BallLoaded_action:
bBallLoaded := TRUE;
END_ACTION

TRANSITION WaitForLifting:
_FBD_ (* Function Block Diagram *)
NETWORK 1
	AND(I_SorterLiftUp, fbDelay.OK)
_END_FBD_
END_TRANSITION
END_ACTION

ACTION BallAvalible_action:
hoBallAvail_ToDS := TRUE;
END_ACTION

ACTION BallRequested_action:
fbDelay(IN_TIME:=tMoveDelay);
END_ACTION

ACTION Transfering_action:
O_SorterGate := TRUE;
fbDelay(IN_TIME:=tTransferDelay);
END_ACTION

ACTION Transfering_exit:
O_SorterGate := FALSE;
END_ACTION

ACTION Unload_Handshake_action:
hoBallAvail_ToDS := FALSE;
END_ACTION

ACTION TransferComplete_action:
bBallLoaded := FALSE;
END_ACTION

ACTION SFCResetStep_action:
SFCReset := TRUE;
END_ACTION
END_FUNCTION_BLOCK

(* POU FBs/FB_Wait, ST *)
FUNCTION_BLOCK FB_Wait
(*Waits the given time and sets output after timer has run till end. When called again timer restarts.
Author: 	Niko Siltala, niko.siltala@tut.fi
Date: 	2014-01-01*)
VAR_INPUT
	IN_TIME	:TIME;		(*Time to wait*)
END_VAR
VAR_OUTPUT
	OK 		: BOOL:=FALSE;	(*Gets true after wait time has expired*)
END_VAR
VAR
	Timer	: TP;
	Falling	: F_TRIG;
END_VAR
IF Timer.Q=TRUE THEN
	(*Call timer block when pulse timer is counting*)
	Timer;
ELSE
	(*Timer has espired. Start it again*)
	Timer(IN:=FALSE);
	Timer(PT:=IN_TIME);
	Timer(IN:=TRUE);
END_IF;
(*Set output. True if timer has expired*)
OK:=NOT Timer.Q;
END_FUNCTION_BLOCK

(* POU FBs/FB_Lift, SFC *)
FUNCTION_BLOCK FB_Lift
VAR_INPUT
	bReset			 : BOOL;	(*Reset Request*)
	bEnable			 : BOOL;
	I_LimitUp 			 : BOOL;
	I_LimitLow 	        : BOOL;
	I_WaitingBallMetal : BOOL;

	(* ColourSensor *)
	I_SenColourYellow		:BOOL;	(*Colour sensor In1 - Yellow*)
	I_SenColourBlue		:BOOL;	(*Colour sensor In2 - Blue*)
	I_SenColourGreen		:BOOL;	(*Colour sensor In3 - Green*)
	I_SenColourRed		:BOOL;	(*Colour sensor In4 - Red*)

	(*SMEMA Handshake Inputs*)
	hiRdyToReceive_FromDS	: BOOL;
	hiBallAvail_FromUS			: BOOL;
END_VAR
VAR_OUTPUT
	bStopOK		: BOOL;
	bBallLoaded	: BOOL;
	bCurBallMetal	: BOOL;
	bCurrentBall 	: E_BallColour := NoColour;

	O_Ejector		:BOOL;

	(*SMEMA Handshake Outputs*)
	hoBallAvail_ToDS				: BOOL;
	hoReadyToRecieve_ToUS	: BOOL;
END_VAR
VAR
	bBallRequested : BOOL := FALSE;
	fbTransferBall	:FB_TransferBall2;

	fbDelay		: FB_Wait;
	tonMoveDelay	: TON;
	tonSensorDelay	: TON;
	tTransferDelay: TIME := T#4s;
	tMoveDelay	: TIME := T#4s;
	tSensorDelay	: TIME := T#2s;
	bLocalReset	: BOOL;	(*Performs local reset*)
	SFCReset 	: BOOL;	(*Resets the execution of SFC to init once this SFCFlag is set true *)
END_VAR
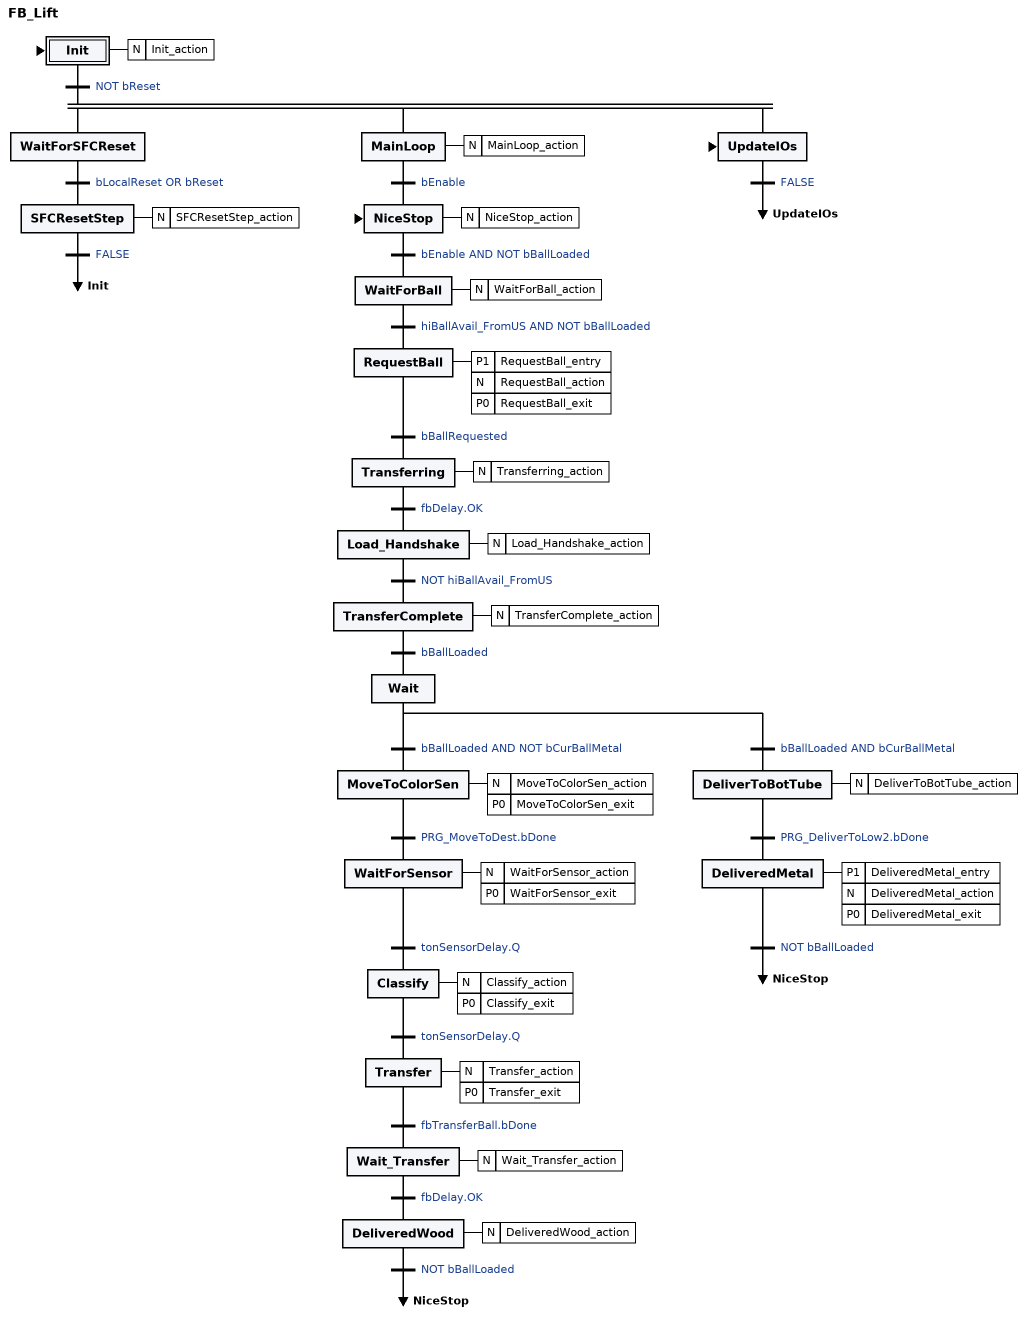
INITIAL_STEP Init:
	Init_action(N);
END_STEP
TRANSITION FROM Init TO (WaitForSFCReset, MainLoop, UpdateIOs) := NOT bReset;
END_TRANSITION
STEP WaitForSFCReset:
END_STEP
TRANSITION FROM WaitForSFCReset TO SFCResetStep := bLocalReset OR bReset;
END_TRANSITION
STEP MainLoop:
	MainLoop_action(N);
END_STEP
TRANSITION FROM MainLoop TO NiceStop := bEnable;
END_TRANSITION
STEP NiceStop:
	NiceStop_action(N);
END_STEP
TRANSITION FROM NiceStop TO WaitForBall := bEnable AND NOT bBallLoaded;
END_TRANSITION
STEP WaitForBall:
	WaitForBall_action(N);
END_STEP
TRANSITION FROM WaitForBall TO RequestBall := hiBallAvail_FromUS AND NOT bBallLoaded;
END_TRANSITION
STEP RequestBall:
	RequestBall_entry(P1);
	RequestBall_action(N);
	RequestBall_exit(P0);
END_STEP
TRANSITION FROM RequestBall TO Transferring := bBallRequested;
END_TRANSITION
STEP Transferring:
	Transferring_action(N);
END_STEP
TRANSITION FROM Transferring TO Load_Handshake := fbDelay.OK;
END_TRANSITION
STEP Load_Handshake:
	Load_Handshake_action(N);
END_STEP
TRANSITION FROM Load_Handshake TO TransferComplete := NOT hiBallAvail_FromUS;
END_TRANSITION
STEP TransferComplete:
	TransferComplete_action(N);
END_STEP
TRANSITION FROM TransferComplete TO Wait := bBallLoaded;
END_TRANSITION
STEP Wait:
END_STEP
TRANSITION FROM Wait TO MoveToColorSen := bBallLoaded AND NOT bCurBallMetal;
END_TRANSITION
TRANSITION FROM Wait TO DeliverToBotTube := bBallLoaded AND bCurBallMetal;
END_TRANSITION
STEP DeliverToBotTube:
	DeliverToBotTube_action(N);
END_STEP
TRANSITION FROM DeliverToBotTube TO DeliveredMetal := PRG_DeliverToLow2.bDone;
END_TRANSITION
STEP DeliveredMetal:
	DeliveredMetal_entry(P1);
	DeliveredMetal_action(N);
	DeliveredMetal_exit(P0);
END_STEP
TRANSITION FROM DeliveredMetal TO NiceStop := NOT bBallLoaded;
END_TRANSITION
STEP MoveToColorSen:
	MoveToColorSen_action(N);
	MoveToColorSen_exit(P0);
END_STEP
TRANSITION FROM MoveToColorSen TO WaitForSensor := PRG_MoveToDest.bDone;
END_TRANSITION
STEP WaitForSensor:
	WaitForSensor_action(N);
	WaitForSensor_exit(P0);
END_STEP
TRANSITION FROM WaitForSensor TO Classify := tonSensorDelay.Q;
END_TRANSITION
STEP Classify:
	Classify_action(N);
	Classify_exit(P0);
END_STEP
TRANSITION FROM Classify TO Transfer := tonSensorDelay.Q;
END_TRANSITION
STEP Transfer:
	Transfer_action(N);
	Transfer_exit(P0);
END_STEP
TRANSITION FROM Transfer TO Wait_Transfer := fbTransferBall.bDone;
END_TRANSITION
STEP Wait_Transfer:
	Wait_Transfer_action(N);
END_STEP
TRANSITION FROM Wait_Transfer TO DeliveredWood := fbDelay.OK;
END_TRANSITION
STEP DeliveredWood:
	DeliveredWood_action(N);
END_STEP
TRANSITION FROM DeliveredWood TO NiceStop := NOT bBallLoaded;
END_TRANSITION
STEP UpdateIOs:
END_STEP
TRANSITION FROM UpdateIOs TO UpdateIOs := FALSE;
END_TRANSITION
STEP SFCResetStep:
	SFCResetStep_action(N);
END_STEP
TRANSITION FROM SFCResetStep TO Init := FALSE;
END_TRANSITION

ACTION Init_action:
SFCReset := FALSE;
bLocalReset	:= FALSE;
END_ACTION

ACTION MainLoop_action:
hoBallAvail_ToDS			  := FALSE;
hoReadyToRecieve_ToUS := FALSE;
END_ACTION

ACTION NiceStop_action:
bStopOK	  	:= TRUE;
bCurrentBall	:= NoColour;
END_ACTION

ACTION WaitForBall_action:
bBallLoaded := FALSE;
hoReadyToRecieve_ToUS := TRUE;
END_ACTION

ACTION RequestBall_entry:
bStopOK := FALSE;
END_ACTION

ACTION RequestBall_action:
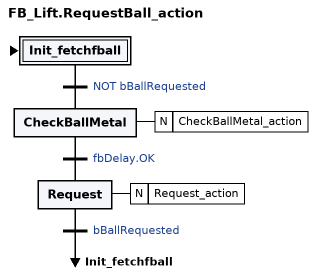
INITIAL_STEP Init_fetchfball:
END_STEP
TRANSITION FROM Init_fetchfball TO CheckBallMetal := NOT bBallRequested;
END_TRANSITION
STEP CheckBallMetal:
	CheckBallMetal_action(N);
END_STEP
TRANSITION FROM CheckBallMetal TO Request := fbDelay.OK;
END_TRANSITION
STEP Request:
	Request_action(N);
END_STEP
TRANSITION FROM Request TO Init_fetchfball := bBallRequested;
END_TRANSITION

ACTION CheckBallMetal_action:
bCurBallMetal	 := I_WaitingBallMetal;
fbDelay(IN_TIME:=T#2s);
END_ACTION

ACTION Request_action:
hoReadyToRecieve_ToUS := TRUE;
bBallRequested := TRUE;
END_ACTION
END_ACTION

ACTION RequestBall_exit:
bBallRequested := FALSE;
END_ACTION

ACTION Transferring_action:
fbDelay(IN_TIME:=tTransferDelay);
END_ACTION

ACTION Load_Handshake_action:
hoReadyToRecieve_ToUS := FALSE;
END_ACTION

ACTION TransferComplete_action:
bBallLoaded := TRUE;
END_ACTION

ACTION DeliverToBotTube_action:
PRG_DeliverToLow2(bExecute:=TRUE ,  bDone=> );
END_ACTION

ACTION DeliveredMetal_entry:
bBallLoaded := FALSE;
PRG_DeliverToLow(bReset:=FALSE , bExecute:=FALSE ,  bDone=> );
END_ACTION

ACTION DeliveredMetal_action:
bBallLoaded := FALSE;
END_ACTION

ACTION DeliveredMetal_exit:
PRG_DeliverToLow(bReset:=FALSE , bExecute:=FALSE ,  bDone=> );
END_ACTION

ACTION MoveToColorSen_action:
PRG_MoveToDest(bExecute:= TRUE, wTarget:= GPOS_COLOR_SEN, bDone:= );
END_ACTION

ACTION MoveToColorSen_exit:
PRG_MoveToDest( bExecute:=FALSE);
END_ACTION

ACTION WaitForSensor_action:
tonSensorDelay(IN:=TRUE , PT:= tSensorDelay);
END_ACTION

ACTION WaitForSensor_exit:
tonSensorDelay(IN:=FALSE);
END_ACTION

ACTION Classify_action:
tonSensorDelay(IN:=TRUE , PT:= tSensorDelay);
IF I_SenColourYellow THEN
	bCurrentBall := Yellow;
ELSIF  I_SenColourBlue THEN
	bCurrentBall := Blue;
ELSIF  I_SenColourRed THEN
	bCurrentBall := Red;
ELSE
	bCurrentBall := NoColour;
END_IF
END_ACTION

ACTION Classify_exit:
tonSensorDelay(IN:=FALSE);
END_ACTION

ACTION Transfer_action:
fbTransferBall(bExecute:= TRUE , bBallToTransfer:= bCurrentBall, bDone=> );
END_ACTION

ACTION Transfer_exit:
fbTransferBall(bExecute:= FALSE);
END_ACTION

ACTION Wait_Transfer_action:
fbDelay(IN_TIME:=tMoveDelay);
END_ACTION

ACTION DeliveredWood_action:
bBallLoaded := FALSE;
bCurrentBall := NoColour;
END_ACTION

ACTION SFCResetStep_action:
SFCReset := TRUE;
END_ACTION
END_FUNCTION_BLOCK

(* POU FBs/FB_TransferBall2, ST *)
FUNCTION_BLOCK FB_TransferBall2
VAR_INPUT
	bExecute			: BOOL;	(*enable and run*)
	bBallToTransfer 	: E_BallColour;
END_VAR
VAR_OUTPUT
	bDone			: BOOL;
	bActDone		: BOOL := FALSE;
END_VAR
VAR
	tonMoveDelay	: TON;
	tonEjectDelay	: TON;
	tMoveDelay	: TIME := T#1s;
	tEjectorDelay	: TIME := T#1s;
END_VAR
IF bExecute THEN
	CASE bBallToTransfer OF
		Yellow:
			PRG_MoveToDest(bExecute:= TRUE , wTarget:= GPOS_PIPE_UP, bDone:= );
			bDone	:= FALSE;
				(*IF PRG_MoveToDest.bDone THEN
					PRG_MoveToDest( bExecute:=FALSE);
					bDone	:= TRUE;
				END_IF*)
		Blue:
			PRG_MoveToDest(bExecute:= TRUE , wTarget:= GPOS_PIPE_MID, bDone:= );
				bDone	:= FALSE;
				(*IF PRG_MoveToDest.bDone THEN
					PRG_MoveToDest( bExecute:=FALSE);
					bDone	:= TRUE;
				END_IF*)
		Red, NoColour:
			PRG_MoveToDest(bExecute:= TRUE , wTarget:= GPOS_GARBAGE, bDone:= );
				bDone	:= FALSE;
				(*IF PRG_MoveToDest.bDone THEN
					PRG_MoveToDest( bExecute:=FALSE);
					bDone	:= TRUE;
				END_IF*)
	ELSE
		PRG_MoveToDest(bExecute:=FALSE);
		bDone	:= FALSE;
	END_CASE

	IF PRG_MoveToDest.bDone THEN
		PRG_MoveToDest(bExecute:=FALSE);
		bDone	:= TRUE;
	END_IF

ELSE
	bDone := FALSE;
END_IF
END_FUNCTION_BLOCK

(* POU Processes/PRG_MoveToDest, SFC *)
PROGRAM PRG_MoveToDest
VAR_INPUT
	bExecute: BOOL;
	wTarget : WORD;
END_VAR
VAR_INPUT
	bDone: BOOL;
END_VAR
VAR
	tonMoveDelay	: TON;
	tonEjectDelay	: TON;
	tonSensorDelay	: TON;
	tMoveDelay		: TIME := T#500ms;
	tEjectorDelay	: TIME := T#1s;
	tSensorDelay	: TIME := T#500ms;
END_VAR
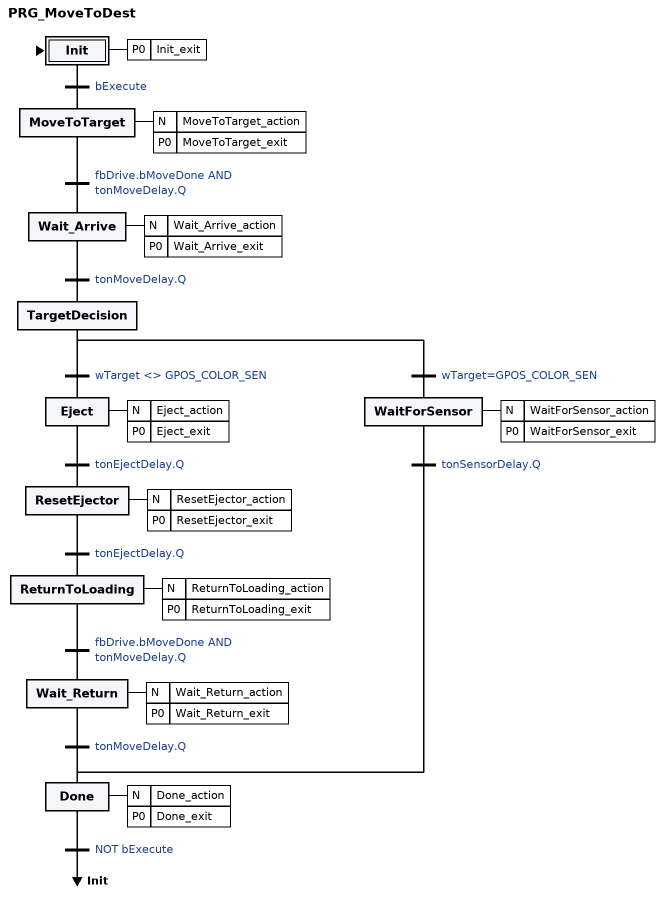
INITIAL_STEP Init:
	Init_exit(P0);
END_STEP
TRANSITION FROM Init TO MoveToTarget := bExecute;
END_TRANSITION
STEP MoveToTarget:
	MoveToTarget_action(N);
	MoveToTarget_exit(P0);
END_STEP
TRANSITION FROM MoveToTarget TO Wait_Arrive := fbDrive.bMoveDone AND tonMoveDelay.Q;
END_TRANSITION
STEP Wait_Arrive:
	Wait_Arrive_action(N);
	Wait_Arrive_exit(P0);
END_STEP
TRANSITION FROM Wait_Arrive TO TargetDecision := tonMoveDelay.Q;
END_TRANSITION
STEP TargetDecision:
END_STEP
TRANSITION FROM TargetDecision TO Eject := wTarget <> GPOS_COLOR_SEN;
END_TRANSITION
TRANSITION FROM TargetDecision TO WaitForSensor := wTarget=GPOS_COLOR_SEN;
END_TRANSITION
STEP WaitForSensor:
	WaitForSensor_action(N);
	WaitForSensor_exit(P0);
END_STEP
TRANSITION FROM WaitForSensor TO Done := tonSensorDelay.Q;
END_TRANSITION
STEP Eject:
	Eject_action(N);
	Eject_exit(P0);
END_STEP
TRANSITION FROM Eject TO ResetEjector := tonEjectDelay.Q;
END_TRANSITION
STEP ResetEjector:
	ResetEjector_action(N);
	ResetEjector_exit(P0);
END_STEP
TRANSITION FROM ResetEjector TO ReturnToLoading := tonEjectDelay.Q;
END_TRANSITION
STEP ReturnToLoading:
	ReturnToLoading_action(N);
	ReturnToLoading_exit(P0);
END_STEP
TRANSITION FROM ReturnToLoading TO Wait_Return := fbDrive.bMoveDone AND tonMoveDelay.Q;
END_TRANSITION
STEP Wait_Return:
	Wait_Return_action(N);
	Wait_Return_exit(P0);
END_STEP
TRANSITION FROM Wait_Return TO Done := tonMoveDelay.Q;
END_TRANSITION
STEP Done:
	Done_action(N);
	Done_exit(P0);
END_STEP
TRANSITION FROM Done TO Init := NOT bExecute;
END_TRANSITION

ACTION Init_exit:
bDone := FALSE;
END_ACTION

ACTION MoveToTarget_action:
tonMoveDelay(IN:=TRUE , PT:= tMoveDelay);
fbDrive(
	bEnable:= TRUE,
	bStart:= TRUE,
	wTarget:= wTarget);
END_ACTION

ACTION MoveToTarget_exit:
fbDrive(
	bStart:= FALSE);
tonMoveDelay(IN:=FALSE);
END_ACTION

ACTION Wait_Arrive_action:
tonMoveDelay(IN:=TRUE , PT:= tMoveDelay);
END_ACTION

ACTION Wait_Arrive_exit:
tonMoveDelay(IN:=FALSE);
END_ACTION

ACTION WaitForSensor_action:
tonSensorDelay(IN:=TRUE , PT:= tSensorDelay);
END_ACTION

ACTION WaitForSensor_exit:
tonSensorDelay(IN:=TRUE , PT:= tSensorDelay);
END_ACTION

ACTION Eject_action:
OEjector := TRUE;
tonEjectDelay(IN:=TRUE , PT:= tEjectorDelay);
END_ACTION

ACTION Eject_exit:
tonEjectDelay(IN:=FALSE);
END_ACTION

ACTION ResetEjector_action:
OEjector := FALSE;
tonEjectDelay(IN:=TRUE , PT:= tEjectorDelay);
END_ACTION

ACTION ResetEjector_exit:
tonEjectDelay(IN:=FALSE);
END_ACTION

ACTION ReturnToLoading_action:
fbDrive(
	bEnable:= TRUE,
	bStart:= TRUE,
	wTarget:= GPOS_LOADING);

tonMoveDelay(IN:=TRUE , PT:= tMoveDelay);
END_ACTION

ACTION ReturnToLoading_exit:
fbDrive(
	bStart:= FALSE);

tonMoveDelay(IN:=FALSE);
END_ACTION

ACTION Wait_Return_action:
tonMoveDelay(IN:=TRUE , PT:= tMoveDelay);
END_ACTION

ACTION Wait_Return_exit:
tonMoveDelay(IN:=FALSE);
END_ACTION

ACTION Done_action:
bDone := TRUE;
END_ACTION

ACTION Done_exit:
bDone := FALSE;
END_ACTION
END_PROGRAM

(* POU OLD/PRG_DeliverToLow2, SFC *)
PROGRAM PRG_DeliverToLow2
VAR_INPUT
	bExecute: BOOL;
END_VAR
VAR_INPUT
	bDone: BOOL;
END_VAR
VAR
	tonMoveDelay	: TON;
	tonEjectDelay	: TON;
	tMoveDelay	: TIME := T#4s;
	tEjectorDelay	: TIME := T#3s;
END_VAR
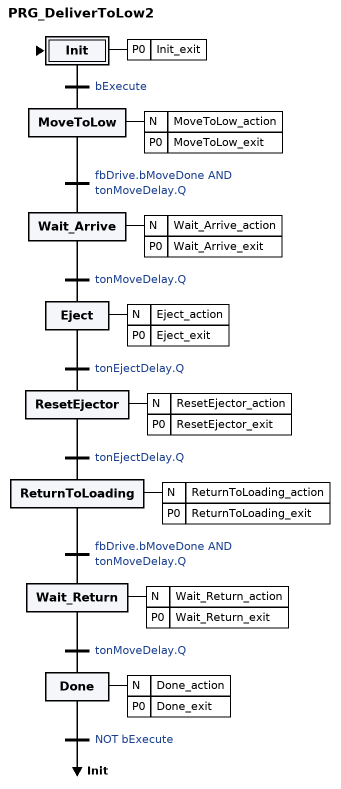
INITIAL_STEP Init:
	Init_exit(P0);
END_STEP
TRANSITION FROM Init TO MoveToLow := bExecute;
END_TRANSITION
STEP MoveToLow:
	MoveToLow_action(N);
	MoveToLow_exit(P0);
END_STEP
TRANSITION FROM MoveToLow TO Wait_Arrive := fbDrive.bMoveDone AND tonMoveDelay.Q;
END_TRANSITION
STEP Wait_Arrive:
	Wait_Arrive_action(N);
	Wait_Arrive_exit(P0);
END_STEP
TRANSITION FROM Wait_Arrive TO Eject := tonMoveDelay.Q;
END_TRANSITION
STEP Eject:
	Eject_action(N);
	Eject_exit(P0);
END_STEP
TRANSITION FROM Eject TO ResetEjector := tonEjectDelay.Q;
END_TRANSITION
STEP ResetEjector:
	ResetEjector_action(N);
	ResetEjector_exit(P0);
END_STEP
TRANSITION FROM ResetEjector TO ReturnToLoading := tonEjectDelay.Q;
END_TRANSITION
STEP ReturnToLoading:
	ReturnToLoading_action(N);
	ReturnToLoading_exit(P0);
END_STEP
TRANSITION FROM ReturnToLoading TO Wait_Return := fbDrive.bMoveDone AND tonMoveDelay.Q;
END_TRANSITION
STEP Wait_Return:
	Wait_Return_action(N);
	Wait_Return_exit(P0);
END_STEP
TRANSITION FROM Wait_Return TO Done := tonMoveDelay.Q;
END_TRANSITION
STEP Done:
	Done_action(N);
	Done_exit(P0);
END_STEP
TRANSITION FROM Done TO Init := NOT bExecute;
END_TRANSITION

ACTION Init_exit:
bDone := FALSE;
END_ACTION

ACTION MoveToLow_action:
tonMoveDelay(IN:=TRUE , PT:= tMoveDelay);
fbDrive(
	bEnable:= TRUE,
	bStart:= TRUE,
	wTarget:= GPOS_PIPE_LOW);
END_ACTION

ACTION MoveToLow_exit:
fbDrive(
	bStart:= FALSE);
tonMoveDelay(IN:=FALSE);
END_ACTION

ACTION Wait_Arrive_action:
tonMoveDelay(IN:=TRUE , PT:= tMoveDelay);
END_ACTION

ACTION Wait_Arrive_exit:
tonMoveDelay(IN:=FALSE);
END_ACTION

ACTION Eject_action:
OEjector := TRUE;
tonEjectDelay(IN:=TRUE , PT:= tEjectorDelay);
END_ACTION

ACTION Eject_exit:
tonEjectDelay(IN:=FALSE);
END_ACTION

ACTION ResetEjector_action:
OEjector := FALSE;
tonEjectDelay(IN:=TRUE , PT:= tEjectorDelay);
END_ACTION

ACTION ResetEjector_exit:
tonEjectDelay(IN:=FALSE);
END_ACTION

ACTION ReturnToLoading_action:
fbDrive(
	bEnable:= TRUE,
	bStart:= TRUE,
	wTarget:= GPOS_LOADING);

tonMoveDelay(IN:=TRUE , PT:= tMoveDelay);
END_ACTION

ACTION ReturnToLoading_exit:
fbDrive(
	bStart:= FALSE);

tonMoveDelay(IN:=FALSE);
END_ACTION

ACTION Wait_Return_action:
tonMoveDelay(IN:=TRUE , PT:= tMoveDelay);
END_ACTION

ACTION Wait_Return_exit:
tonMoveDelay(IN:=FALSE);
END_ACTION

ACTION Done_action:
bDone := TRUE;
END_ACTION

ACTION Done_exit:
bDone := FALSE;
END_ACTION
END_PROGRAM

(* POU OLD/PRG_DeliverToLow, SFC *)
PROGRAM PRG_DeliverToLow
VAR_INPUT
	bReset		: BOOL;	(*Reset program*)
	bExecute		: BOOL;	(*enable and run*)

END_VAR
VAR_OUTPUT
	bDone			: BOOL;
END_VAR
VAR
	tonMoveDelay	: TON;
	tonEjectDelay	: TON;
	SFCReset		: BOOL;

	tMoveDelay	: TIME := T#4s;
	tEjectorDelay	: TIME := T#3s;
END_VAR
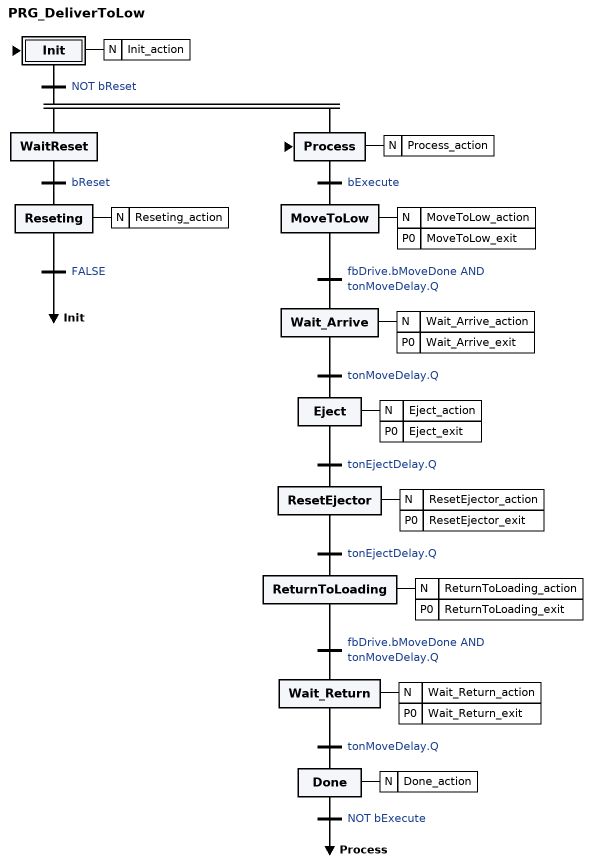
INITIAL_STEP Init:
	Init_action(N);
END_STEP
TRANSITION FROM Init TO (WaitReset, Process) := NOT bReset;
END_TRANSITION
STEP WaitReset:
END_STEP
TRANSITION FROM WaitReset TO Reseting := bReset;
END_TRANSITION
STEP Process:
	Process_action(N);
END_STEP
TRANSITION FROM Process TO MoveToLow := bExecute;
END_TRANSITION
STEP MoveToLow:
	MoveToLow_action(N);
	MoveToLow_exit(P0);
END_STEP
TRANSITION FROM MoveToLow TO Wait_Arrive := fbDrive.bMoveDone AND tonMoveDelay.Q;
END_TRANSITION
STEP Wait_Arrive:
	Wait_Arrive_action(N);
	Wait_Arrive_exit(P0);
END_STEP
TRANSITION FROM Wait_Arrive TO Eject := tonMoveDelay.Q;
END_TRANSITION
STEP Eject:
	Eject_action(N);
	Eject_exit(P0);
END_STEP
TRANSITION FROM Eject TO ResetEjector := tonEjectDelay.Q;
END_TRANSITION
STEP ResetEjector:
	ResetEjector_action(N);
	ResetEjector_exit(P0);
END_STEP
TRANSITION FROM ResetEjector TO ReturnToLoading := tonEjectDelay.Q;
END_TRANSITION
STEP ReturnToLoading:
	ReturnToLoading_action(N);
	ReturnToLoading_exit(P0);
END_STEP
TRANSITION FROM ReturnToLoading TO Wait_Return := fbDrive.bMoveDone AND tonMoveDelay.Q;
END_TRANSITION
STEP Wait_Return:
	Wait_Return_action(N);
	Wait_Return_exit(P0);
END_STEP
TRANSITION FROM Wait_Return TO Done := tonMoveDelay.Q;
END_TRANSITION
STEP Done:
	Done_action(N);
END_STEP
TRANSITION FROM Done TO Process := NOT bExecute;
END_TRANSITION
STEP Reseting:
	Reseting_action(N);
END_STEP
TRANSITION FROM Reseting TO Init := FALSE;
END_TRANSITION

ACTION Init_action:
SFCReset := FALSE;
bDone := FALSE;
END_ACTION

ACTION Process_action:
bDone := FALSE;
END_ACTION

ACTION MoveToLow_action:
bDone := FALSE;

fbDrive(
	bEnable:= TRUE,
	bStart:= TRUE,
	wTarget:= GPOS_PIPE_LOW);

tonMoveDelay(IN:=TRUE , PT:= tMoveDelay);
END_ACTION

ACTION MoveToLow_exit:
fbDrive(
	bStart:= FALSE);
tonMoveDelay(IN:=FALSE);
END_ACTION

ACTION Wait_Arrive_action:
tonMoveDelay(IN:=TRUE , PT:= tMoveDelay);
END_ACTION

ACTION Wait_Arrive_exit:
tonMoveDelay(IN:=FALSE);
END_ACTION

ACTION Eject_action:
OEjector := TRUE;
tonEjectDelay(IN:=TRUE , PT:= tEjectorDelay);
END_ACTION

ACTION Eject_exit:
tonEjectDelay(IN:=FALSE);
END_ACTION

ACTION ResetEjector_action:
OEjector := FALSE;
tonEjectDelay(IN:=TRUE , PT:= tEjectorDelay);
END_ACTION

ACTION ResetEjector_exit:
tonEjectDelay(IN:=FALSE);
END_ACTION

ACTION ReturnToLoading_action:
fbDrive(
	bEnable:= TRUE,
	bStart:= TRUE,
	wTarget:= GPOS_LOADING);

tonMoveDelay(IN:=TRUE , PT:= tMoveDelay);
END_ACTION

ACTION ReturnToLoading_exit:
fbDrive(
	bStart:= FALSE);

tonMoveDelay(IN:=FALSE);
END_ACTION

ACTION Wait_Return_action:
tonMoveDelay(IN:=TRUE , PT:= tMoveDelay);
END_ACTION

ACTION Wait_Return_exit:
tonMoveDelay(IN:=FALSE);
END_ACTION

ACTION Done_action:
bDone := TRUE;
END_ACTION

ACTION Reseting_action:
SFCReset := TRUE;
END_ACTION
END_PROGRAM

(* POU Programs/PRG_Drive_Link, FBD *)
PROGRAM PRG_Drive_Link
VAR
END_VAR
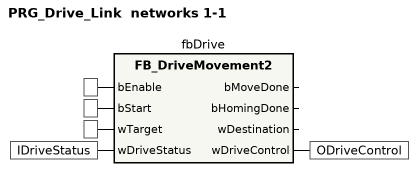
_FBD_ (* Function Block Diagram *)
NETWORK 1
	fbDrive:FB_DriveMovement2(bEnable: , bStart: , wTarget: , wDriveStatus: IDriveStatus, wDriveControl => ODriveControl)
_END_FBD_
END_PROGRAM

(* POU FBs/FB_DriveMovement2, ST *)
FUNCTION_BLOCK FB_DriveMovement2
(* This function block is making all movements for the drive
	bEnable = must be TRUE
	Target = int value of 0 - 63
	bStart = with rising edge starts the movement

	bMoveDone gets true when the movement is finalised.
Author: 	Niko Siltala, niko.siltala@tut.fi
Date: 	2014-01-01*)

VAR_INPUT
	bEnable			: BOOL:=FALSE;	(*Enables the fuction block*)
	bStart			: BOOL:=FALSE;	(*Starts the motion to target by rising edge*)
	wTarget			: WORD:=0;		(*Target destination*)
	wDriveStatus		: WORD;			(*Status word from Indramat Drive*)
END_VAR
VAR_OUTPUT
	bMoveDone		:BOOL:=FALSE;	(*The commanded move has been completed. Drive is at required destination*)
	bHomingDone	:BOOL:=FALSE;	(*Drive has been homed*)
	wDestination		:WORD;			(*Current destination*)
	wDriveControl		:WORD;			(*Control word to Indramat Drive*)
END_VAR
VAR_IN_OUT
END_VAR
VAR
	TONTimer1 	: TON;
	TONTimer2 	: TON;
END_VAR
(*
This function block is making all movements for the drive
	bEnable = must be TRUE
	Target = int value of 0 - 63
	bStart = with rising edge starts the movement

	bMoveDone gets true when the movement is finalised
*)
IF bEnable THEN
	(*Drive is Enabled*)
	wDriveControl:=wDriveControl OR 16#0001;
	IF (wDriveStatus AND 16#0080)>0 AND (wDriveStatus AND 16#0040)>0 THEN
		IF bStart=TRUE THEN
			(*bStart is true*)
			IF bHomingDone=FALSE THEN
				(*Homing procedure*)
				IF TONTimer1.Q=FALSE THEN
					wDriveControl:=16#0005;
					TONTimer1(IN:=TRUE, PT:=T#100ms);(*100ms*)
				ELSE
					IF TONTimer2.Q=FALSE THEN
						(*Start drive*)
						wDriveControl:=16#0007;
						TONTimer2(IN:=TRUE, PT:=T#500ms); (*500ms*)
					ELSE
						(*Timer2 have expired*)
						IF (wDriveStatus AND 16#0004)>0 THEN
							TONTimer1(IN:=FALSE);
							TONTimer2(IN:=FALSE);
							wDriveControl:=16#0001;
							bHomingDone:=TRUE;
						END_IF;
					END_IF;
				END_IF;
			ELSE
				(*Normal movement*)
				IF TONTimer1.Q=FALSE THEN
					(*Set target and Enabled*)
					wDriveControl:=SHL(wTarget,8) OR 16#0001;
					wDestination:=wTarget;
					TONTimer1(IN:=TRUE, PT:=T#10ms);(*10ms*)
				ELSE
					IF TONTimer2.Q=FALSE THEN
						(*Start drive*)
						wDriveControl:=wDriveControl OR 16#0002;
						TONTimer2(IN:=TRUE, PT:=T#500ms); (*500ms*)
					ELSE
						(*Timer2 have expired*)
						IF (wDriveStatus AND 16#0010)>0 THEN
							(*End the movement when user forgets to provide lowering edge*)
							(*bStart:=FALSE;*)
							(*Requested movement is done*)
							bMoveDone:=TRUE;
						END_IF;
					END_IF;
				END_IF; (*Normal movement*)
			END_IF;(*bHomingDone=FALSE*)
		ELSE
			(*bStart is false*)
			bMoveDone:=FALSE;
			TONTimer1(IN:=FALSE);
			TONTimer2(IN:=FALSE);
		END_IF;
	END_IF;
ELSE (*bEnable*)
	(*Drive is NOT Enabled*)
	wDriveControl:=16#0000;
	bMoveDone:=FALSE;
	bHomingDone:=FALSE;
	TONTimer1(IN:=FALSE);
	TONTimer2(IN:=FALSE);
END_IF;
END_FUNCTION_BLOCK

(* POU EXAMPLES, SFC *)
PROGRAM EXAMPLES
VAR
	fbDrive			: DriveMovement2;		(*FB for executing the motion*)
	tonTimer			: TON;			(*Standard TON timer. Use this*)
	fbDelay			: FB_Wait;		(*Different simplified timer.
END_VAR
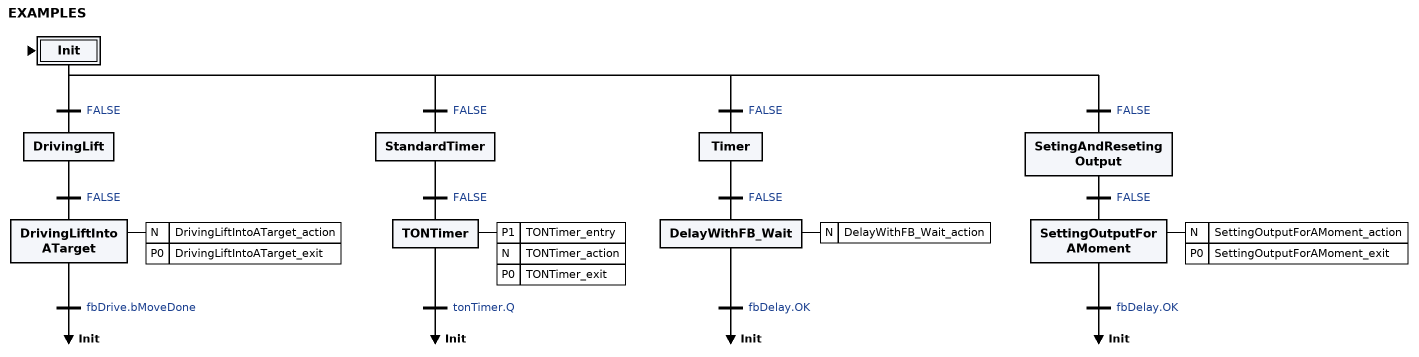
INITIAL_STEP Init:
END_STEP
TRANSITION FROM Init TO DrivingLift := FALSE;
END_TRANSITION
TRANSITION FROM Init TO StandardTimer := FALSE;
END_TRANSITION
TRANSITION FROM Init TO Timer := FALSE;
END_TRANSITION
TRANSITION FROM Init TO SetingAndResetingOutput := FALSE;
END_TRANSITION
STEP DrivingLift:
END_STEP
TRANSITION FROM DrivingLift TO DrivingLiftIntoATarget := FALSE;
END_TRANSITION
STEP DrivingLiftIntoATarget:
	DrivingLiftIntoATarget_action(N);
	DrivingLiftIntoATarget_exit(P0);
END_STEP
TRANSITION FROM DrivingLiftIntoATarget TO Init := fbDrive.bMoveDone;
END_TRANSITION
STEP StandardTimer:
END_STEP
TRANSITION FROM StandardTimer TO TONTimer := FALSE;
END_TRANSITION
STEP TONTimer:
	TONTimer_entry(P1);
	TONTimer_action(N);
	TONTimer_exit(P0);
END_STEP
TRANSITION FROM TONTimer TO Init := tonTimer.Q;
END_TRANSITION
STEP Timer:
END_STEP
TRANSITION FROM Timer TO DelayWithFB_Wait := FALSE;
END_TRANSITION
STEP DelayWithFB_Wait:
	DelayWithFB_Wait_action(N);
END_STEP
TRANSITION FROM DelayWithFB_Wait TO Init := fbDelay.OK;
END_TRANSITION
STEP SetingAndResetingOutput:
END_STEP
TRANSITION FROM SetingAndResetingOutput TO SettingOutputForAMoment := FALSE;
END_TRANSITION
STEP SettingOutputForAMoment:
	SettingOutputForAMoment_action(N);
	SettingOutputForAMoment_exit(P0);
END_STEP
TRANSITION FROM SettingOutputForAMoment TO Init := fbDelay.OK;
END_TRANSITION

ACTION DrivingLiftIntoATarget_action:
(*This executes and drives the lift to desired level (=wTarget)
wTarget is selected from given constants. See:Global Constants*)
fbDrive(
	bEnable:= TRUE,
	bStart:= TRUE,
	wTarget:= GPOS_LOADING);
END_ACTION

ACTION DrivingLiftIntoATarget_exit:
(*Stops the motion*)
fbDrive(
	bStart:= FALSE);
END_ACTION

ACTION TONTimer_entry:
tonTimer(IN:=FALSE);
END_ACTION

ACTION TONTimer_action:
tonTimer(IN:=TRUE , PT:=T#1s, Q=> , ET=> );
END_ACTION

ACTION TONTimer_exit:
tonTimer(IN:=FALSE);
END_ACTION

ACTION DelayWithFB_Wait_action:
(*Timer is counting*)
fbDelay(IN_TIME:=T#1s);
END_ACTION

ACTION SettingOutputForAMoment_action:
(*Timer is counting*)
fbDelay(IN_TIME:=T#500ms);

(*Setting Output*)
OEjector := TRUE;
END_ACTION

ACTION SettingOutputForAMoment_exit:
(*Clearing Output*)
OEjector := FALSE;
END_ACTION
END_PROGRAM

(* POU OLD/PRG_DeliverToGarbage, SFC *)
PROGRAM PRG_DeliverToGarbage
VAR_INPUT
	bReset		: BOOL;	(*Reset program*)
	bExecute		: BOOL;	(*enable and run*)
END_VAR
VAR_OUTPUT
	bDone			: BOOL;
END_VAR
VAR
	tonMoveDelay	: TON;
	tonEjectDelay	: TON;
	SFCReset		: BOOL;

	tMoveDelay	: TIME := T#4s;
	tEjectorDelay	: TIME := T#2s;
END_VAR
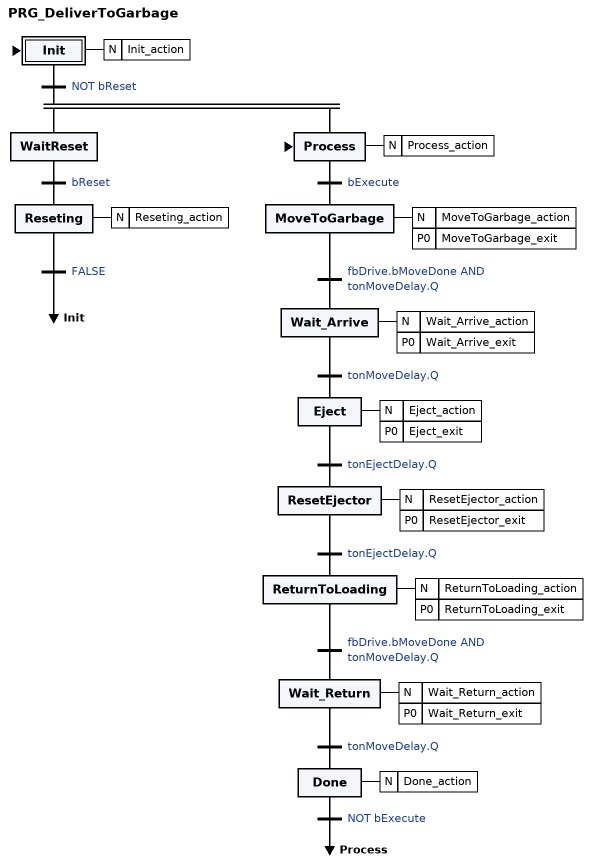
INITIAL_STEP Init:
	Init_action(N);
END_STEP
TRANSITION FROM Init TO (WaitReset, Process) := NOT bReset;
END_TRANSITION
STEP WaitReset:
END_STEP
TRANSITION FROM WaitReset TO Reseting := bReset;
END_TRANSITION
STEP Process:
	Process_action(N);
END_STEP
TRANSITION FROM Process TO MoveToGarbage := bExecute;
END_TRANSITION
STEP MoveToGarbage:
	MoveToGarbage_action(N);
	MoveToGarbage_exit(P0);
END_STEP
TRANSITION FROM MoveToGarbage TO Wait_Arrive := fbDrive.bMoveDone AND tonMoveDelay.Q;
END_TRANSITION
STEP Wait_Arrive:
	Wait_Arrive_action(N);
	Wait_Arrive_exit(P0);
END_STEP
TRANSITION FROM Wait_Arrive TO Eject := tonMoveDelay.Q;
END_TRANSITION
STEP Eject:
	Eject_action(N);
	Eject_exit(P0);
END_STEP
TRANSITION FROM Eject TO ResetEjector := tonEjectDelay.Q;
END_TRANSITION
STEP ResetEjector:
	ResetEjector_action(N);
	ResetEjector_exit(P0);
END_STEP
TRANSITION FROM ResetEjector TO ReturnToLoading := tonEjectDelay.Q;
END_TRANSITION
STEP ReturnToLoading:
	ReturnToLoading_action(N);
	ReturnToLoading_exit(P0);
END_STEP
TRANSITION FROM ReturnToLoading TO Wait_Return := fbDrive.bMoveDone AND tonMoveDelay.Q;
END_TRANSITION
STEP Wait_Return:
	Wait_Return_action(N);
	Wait_Return_exit(P0);
END_STEP
TRANSITION FROM Wait_Return TO Done := tonMoveDelay.Q;
END_TRANSITION
STEP Done:
	Done_action(N);
END_STEP
TRANSITION FROM Done TO Process := NOT bExecute;
END_TRANSITION
STEP Reseting:
	Reseting_action(N);
END_STEP
TRANSITION FROM Reseting TO Init := FALSE;
END_TRANSITION

ACTION Init_action:
SFCReset := FALSE;
bDone := FALSE;
END_ACTION

ACTION Process_action:
bDone := FALSE;
END_ACTION

ACTION MoveToGarbage_action:
bDone := FALSE;

fbDrive(
	bEnable:= TRUE,
	bStart:= TRUE,
	wTarget:= GPOS_GARBAGE);

tonMoveDelay(IN:=TRUE , PT:= tMoveDelay);
END_ACTION

ACTION MoveToGarbage_exit:
fbDrive(
	bStart:= FALSE);

tonMoveDelay(IN:=FALSE);
END_ACTION

ACTION Wait_Arrive_action:
tonMoveDelay(IN:=TRUE , PT:= tMoveDelay);
END_ACTION

ACTION Wait_Arrive_exit:
tonMoveDelay(IN:=FALSE);
END_ACTION

ACTION Eject_action:
OEjector := TRUE;
tonEjectDelay(IN:=TRUE , PT:= tEjectorDelay);
END_ACTION

ACTION Eject_exit:
tonEjectDelay(IN:=FALSE);
END_ACTION

ACTION ResetEjector_action:
OEjector := FALSE;
tonEjectDelay(IN:=TRUE , PT:= tEjectorDelay);
END_ACTION

ACTION ResetEjector_exit:
tonEjectDelay(IN:=FALSE);
END_ACTION

ACTION ReturnToLoading_action:
fbDrive(
	bEnable:= TRUE,
	bStart:= TRUE,
	wTarget:= GPOS_LOADING);

tonMoveDelay(IN:=TRUE , PT:= tMoveDelay);
END_ACTION

ACTION ReturnToLoading_exit:
fbDrive(
	bStart:= FALSE);

tonMoveDelay(IN:=FALSE);
END_ACTION

ACTION Wait_Return_action:
tonMoveDelay(IN:=TRUE , PT:= tMoveDelay);
END_ACTION

ACTION Wait_Return_exit:
tonMoveDelay(IN:=FALSE);
END_ACTION

ACTION Done_action:
bDone := TRUE;
END_ACTION

ACTION Reseting_action:
SFCReset := TRUE;
END_ACTION
END_PROGRAM

(* POU OLD/PRG_DeliverToGarbage2, SFC *)
PROGRAM PRG_DeliverToGarbage2
VAR_INPUT
	bExecute: BOOL;
END_VAR
VAR_INPUT
	bDone: BOOL;
END_VAR
VAR
	tonMoveDelay	: TON;
	tonEjectDelay	: TON;
	tMoveDelay	: TIME := T#3s;
	tEjectorDelay	: TIME := T#3s;
END_VAR
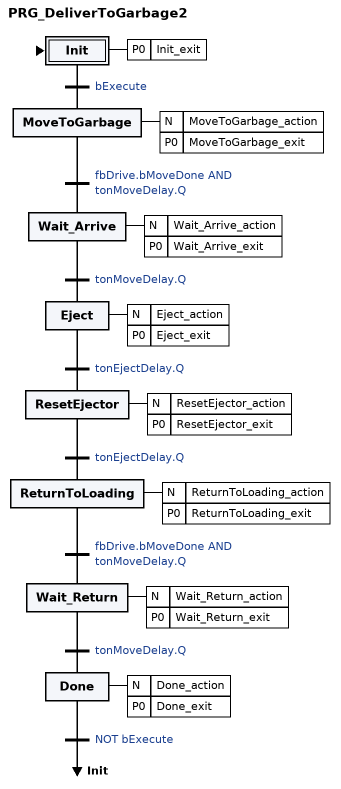
INITIAL_STEP Init:
	Init_exit(P0);
END_STEP
TRANSITION FROM Init TO MoveToGarbage := bExecute;
END_TRANSITION
STEP MoveToGarbage:
	MoveToGarbage_action(N);
	MoveToGarbage_exit(P0);
END_STEP
TRANSITION FROM MoveToGarbage TO Wait_Arrive := fbDrive.bMoveDone AND tonMoveDelay.Q;
END_TRANSITION
STEP Wait_Arrive:
	Wait_Arrive_action(N);
	Wait_Arrive_exit(P0);
END_STEP
TRANSITION FROM Wait_Arrive TO Eject := tonMoveDelay.Q;
END_TRANSITION
STEP Eject:
	Eject_action(N);
	Eject_exit(P0);
END_STEP
TRANSITION FROM Eject TO ResetEjector := tonEjectDelay.Q;
END_TRANSITION
STEP ResetEjector:
	ResetEjector_action(N);
	ResetEjector_exit(P0);
END_STEP
TRANSITION FROM ResetEjector TO ReturnToLoading := tonEjectDelay.Q;
END_TRANSITION
STEP ReturnToLoading:
	ReturnToLoading_action(N);
	ReturnToLoading_exit(P0);
END_STEP
TRANSITION FROM ReturnToLoading TO Wait_Return := fbDrive.bMoveDone AND tonMoveDelay.Q;
END_TRANSITION
STEP Wait_Return:
	Wait_Return_action(N);
	Wait_Return_exit(P0);
END_STEP
TRANSITION FROM Wait_Return TO Done := tonMoveDelay.Q;
END_TRANSITION
STEP Done:
	Done_action(N);
	Done_exit(P0);
END_STEP
TRANSITION FROM Done TO Init := NOT bExecute;
END_TRANSITION

ACTION Init_exit:
bDone := FALSE;
END_ACTION

ACTION MoveToGarbage_action:
fbDrive(
	bEnable:= TRUE,
	bStart:= TRUE,
	wTarget:= GPOS_GARBAGE);

tonMoveDelay(IN:=TRUE , PT:= tMoveDelay);
END_ACTION

ACTION MoveToGarbage_exit:
fbDrive(
	bStart:= FALSE);
tonMoveDelay(IN:=FALSE);
END_ACTION

ACTION Wait_Arrive_action:
tonMoveDelay(IN:=TRUE , PT:= tMoveDelay);
END_ACTION

ACTION Wait_Arrive_exit:
tonMoveDelay(IN:=FALSE);
END_ACTION

ACTION Eject_action:
OEjector := TRUE;
tonEjectDelay(IN:=TRUE , PT:= tEjectorDelay);
END_ACTION

ACTION Eject_exit:
tonEjectDelay(IN:=FALSE);
END_ACTION

ACTION ResetEjector_action:
OEjector := FALSE;
tonEjectDelay(IN:=TRUE , PT:= tEjectorDelay);
END_ACTION

ACTION ResetEjector_exit:
tonEjectDelay(IN:=FALSE);
END_ACTION

ACTION ReturnToLoading_action:
fbDrive(
	bEnable:= TRUE,
	bStart:= TRUE,
	wTarget:= GPOS_LOADING);

tonMoveDelay(IN:=TRUE , PT:= tMoveDelay);
END_ACTION

ACTION ReturnToLoading_exit:
fbDrive(
	bStart:= FALSE);

tonMoveDelay(IN:=FALSE);
END_ACTION

ACTION Wait_Return_action:
tonMoveDelay(IN:=TRUE , PT:= tMoveDelay);
END_ACTION

ACTION Wait_Return_exit:
tonMoveDelay(IN:=FALSE);
END_ACTION

ACTION Done_action:
bDone := TRUE;
END_ACTION

ACTION Done_exit:
bDone := FALSE;
END_ACTION
END_PROGRAM

(* POU OLD/PRG_DeliverToMid, SFC *)
PROGRAM PRG_DeliverToMid
VAR_INPUT
	bReset		: BOOL;	(*Reset program*)
	bExecute		: BOOL;	(*enable and run*)
END_VAR
VAR_OUTPUT
	bDone			: BOOL;
END_VAR
VAR
	tonMoveDelay	: TON;
	tonEjectDelay	: TON;
	SFCReset		: BOOL;

	tMoveDelay	: TIME := T#4s;
	tEjectorDelay	: TIME := T#2s;
END_VAR
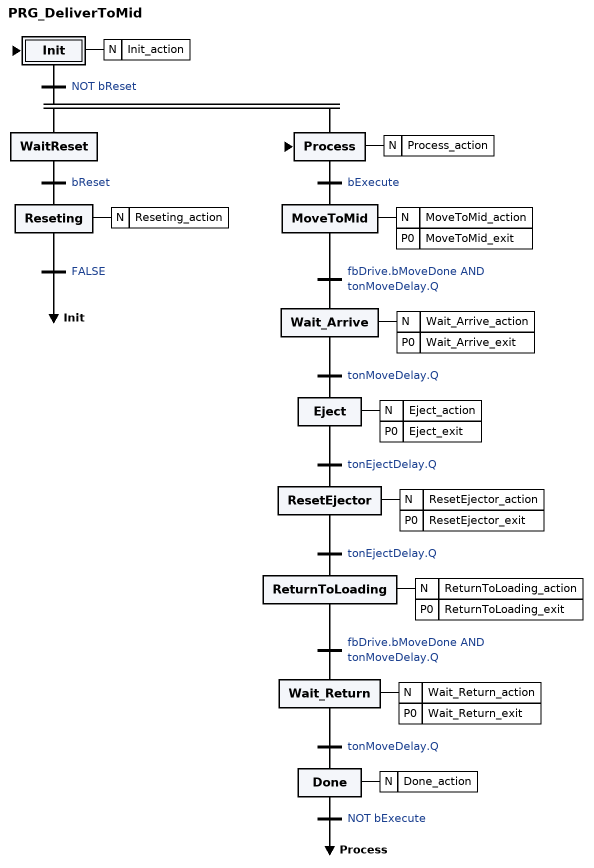
INITIAL_STEP Init:
	Init_action(N);
END_STEP
TRANSITION FROM Init TO (WaitReset, Process) := NOT bReset;
END_TRANSITION
STEP WaitReset:
END_STEP
TRANSITION FROM WaitReset TO Reseting := bReset;
END_TRANSITION
STEP Process:
	Process_action(N);
END_STEP
TRANSITION FROM Process TO MoveToMid := bExecute;
END_TRANSITION
STEP MoveToMid:
	MoveToMid_action(N);
	MoveToMid_exit(P0);
END_STEP
TRANSITION FROM MoveToMid TO Wait_Arrive := fbDrive.bMoveDone AND tonMoveDelay.Q;
END_TRANSITION
STEP Wait_Arrive:
	Wait_Arrive_action(N);
	Wait_Arrive_exit(P0);
END_STEP
TRANSITION FROM Wait_Arrive TO Eject := tonMoveDelay.Q;
END_TRANSITION
STEP Eject:
	Eject_action(N);
	Eject_exit(P0);
END_STEP
TRANSITION FROM Eject TO ResetEjector := tonEjectDelay.Q;
END_TRANSITION
STEP ResetEjector:
	ResetEjector_action(N);
	ResetEjector_exit(P0);
END_STEP
TRANSITION FROM ResetEjector TO ReturnToLoading := tonEjectDelay.Q;
END_TRANSITION
STEP ReturnToLoading:
	ReturnToLoading_action(N);
	ReturnToLoading_exit(P0);
END_STEP
TRANSITION FROM ReturnToLoading TO Wait_Return := fbDrive.bMoveDone AND tonMoveDelay.Q;
END_TRANSITION
STEP Wait_Return:
	Wait_Return_action(N);
	Wait_Return_exit(P0);
END_STEP
TRANSITION FROM Wait_Return TO Done := tonMoveDelay.Q;
END_TRANSITION
STEP Done:
	Done_action(N);
END_STEP
TRANSITION FROM Done TO Process := NOT bExecute;
END_TRANSITION
STEP Reseting:
	Reseting_action(N);
END_STEP
TRANSITION FROM Reseting TO Init := FALSE;
END_TRANSITION

ACTION Init_action:
SFCReset := FALSE;
bDone := FALSE;
END_ACTION

ACTION Process_action:
bDone := FALSE;
END_ACTION

ACTION MoveToMid_action:
bDone := FALSE;

fbDrive(
	bEnable:= TRUE,
	bStart:= TRUE,
	wTarget:=GPOS_PIPE_MID);

tonMoveDelay(IN:=TRUE , PT:= tMoveDelay);
END_ACTION

ACTION MoveToMid_exit:
fbDrive(
	bStart:= FALSE);

tonMoveDelay(IN:=FALSE);
END_ACTION

ACTION Wait_Arrive_action:
tonMoveDelay(IN:=TRUE , PT:= tMoveDelay);
END_ACTION

ACTION Wait_Arrive_exit:
tonMoveDelay(IN:=FALSE);
END_ACTION

ACTION Eject_action:
OEjector := TRUE;
tonEjectDelay(IN:=TRUE , PT:= tEjectorDelay);
END_ACTION

ACTION Eject_exit:
tonEjectDelay(IN:=FALSE);
END_ACTION

ACTION ResetEjector_action:
OEjector := FALSE;
tonEjectDelay(IN:=TRUE , PT:= tEjectorDelay);
END_ACTION

ACTION ResetEjector_exit:
tonEjectDelay(IN:=FALSE);
END_ACTION

ACTION ReturnToLoading_action:
fbDrive(
	bEnable:= TRUE,
	bStart:= TRUE,
	wTarget:= GPOS_LOADING);

tonMoveDelay(IN:=TRUE , PT:= tMoveDelay);
END_ACTION

ACTION ReturnToLoading_exit:
fbDrive(
	bStart:= FALSE);

tonMoveDelay(IN:=FALSE);
END_ACTION

ACTION Wait_Return_action:
tonMoveDelay(IN:=TRUE , PT:= tMoveDelay);
END_ACTION

ACTION Wait_Return_exit:
tonMoveDelay(IN:=FALSE);
END_ACTION

ACTION Done_action:
bDone := TRUE;
END_ACTION

ACTION Reseting_action:
SFCReset := TRUE;
END_ACTION
END_PROGRAM

(* POU OLD/PRG_DeliverToMid2, SFC *)
PROGRAM PRG_DeliverToMid2
VAR_INPUT
	bExecute: BOOL;
END_VAR
VAR_INPUT
	bDone: BOOL;
END_VAR
VAR
	tonMoveDelay	: TON;
	tonEjectDelay	: TON;
	tMoveDelay	: TIME := T#3s;
	tEjectorDelay	: TIME := T#3s;
END_VAR
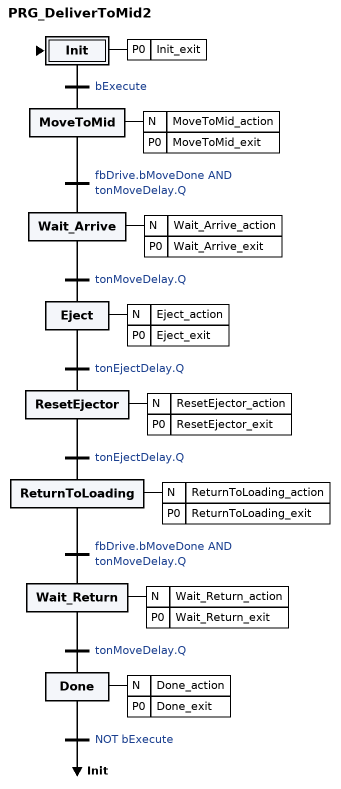
INITIAL_STEP Init:
	Init_exit(P0);
END_STEP
TRANSITION FROM Init TO MoveToMid := bExecute;
END_TRANSITION
STEP MoveToMid:
	MoveToMid_action(N);
	MoveToMid_exit(P0);
END_STEP
TRANSITION FROM MoveToMid TO Wait_Arrive := fbDrive.bMoveDone AND tonMoveDelay.Q;
END_TRANSITION
STEP Wait_Arrive:
	Wait_Arrive_action(N);
	Wait_Arrive_exit(P0);
END_STEP
TRANSITION FROM Wait_Arrive TO Eject := tonMoveDelay.Q;
END_TRANSITION
STEP Eject:
	Eject_action(N);
	Eject_exit(P0);
END_STEP
TRANSITION FROM Eject TO ResetEjector := tonEjectDelay.Q;
END_TRANSITION
STEP ResetEjector:
	ResetEjector_action(N);
	ResetEjector_exit(P0);
END_STEP
TRANSITION FROM ResetEjector TO ReturnToLoading := tonEjectDelay.Q;
END_TRANSITION
STEP ReturnToLoading:
	ReturnToLoading_action(N);
	ReturnToLoading_exit(P0);
END_STEP
TRANSITION FROM ReturnToLoading TO Wait_Return := fbDrive.bMoveDone AND tonMoveDelay.Q;
END_TRANSITION
STEP Wait_Return:
	Wait_Return_action(N);
	Wait_Return_exit(P0);
END_STEP
TRANSITION FROM Wait_Return TO Done := tonMoveDelay.Q;
END_TRANSITION
STEP Done:
	Done_action(N);
	Done_exit(P0);
END_STEP
TRANSITION FROM Done TO Init := NOT bExecute;
END_TRANSITION

ACTION Init_exit:
bDone := FALSE;
END_ACTION

ACTION MoveToMid_action:
fbDrive(
	bEnable:= TRUE,
	bStart:= TRUE,
	wTarget:= GPOS_PIPE_MID);

tonMoveDelay(IN:=TRUE , PT:= tMoveDelay);
END_ACTION

ACTION MoveToMid_exit:
fbDrive(
	bStart:= FALSE);
tonMoveDelay(IN:=FALSE);
END_ACTION

ACTION Wait_Arrive_action:
tonMoveDelay(IN:=TRUE , PT:= tMoveDelay);
END_ACTION

ACTION Wait_Arrive_exit:
tonMoveDelay(IN:=FALSE);
END_ACTION

ACTION Eject_action:
OEjector := TRUE;
tonEjectDelay(IN:=TRUE , PT:= tEjectorDelay);
END_ACTION

ACTION Eject_exit:
tonEjectDelay(IN:=FALSE);
END_ACTION

ACTION ResetEjector_action:
OEjector := FALSE;
tonEjectDelay(IN:=TRUE , PT:= tEjectorDelay);
END_ACTION

ACTION ResetEjector_exit:
tonEjectDelay(IN:=FALSE);
END_ACTION

ACTION ReturnToLoading_action:
fbDrive(
	bEnable:= TRUE,
	bStart:= TRUE,
	wTarget:= GPOS_LOADING);

tonMoveDelay(IN:=TRUE , PT:= tMoveDelay);
END_ACTION

ACTION ReturnToLoading_exit:
fbDrive(
	bStart:= FALSE);

tonMoveDelay(IN:=FALSE);
END_ACTION

ACTION Wait_Return_action:
tonMoveDelay(IN:=TRUE , PT:= tMoveDelay);
END_ACTION

ACTION Wait_Return_exit:
tonMoveDelay(IN:=FALSE);
END_ACTION

ACTION Done_action:
bDone := TRUE;
END_ACTION

ACTION Done_exit:
bDone := FALSE;
END_ACTION
END_PROGRAM

(* POU OLD/PRG_DeliverToUp, SFC *)
PROGRAM PRG_DeliverToUp
VAR_INPUT
	bReset		: BOOL;	(*Reset program*)
	bExecute		: BOOL;	(*enable and run*)
END_VAR
VAR_OUTPUT
	bDone			: BOOL;
END_VAR
VAR
	tonMoveDelay	: TON;
	tonEjectDelay	: TON;
	SFCReset		: BOOL;

	tMoveDelay	: TIME := T#4s;
	tEjectorDelay	: TIME := T#2s;
END_VAR
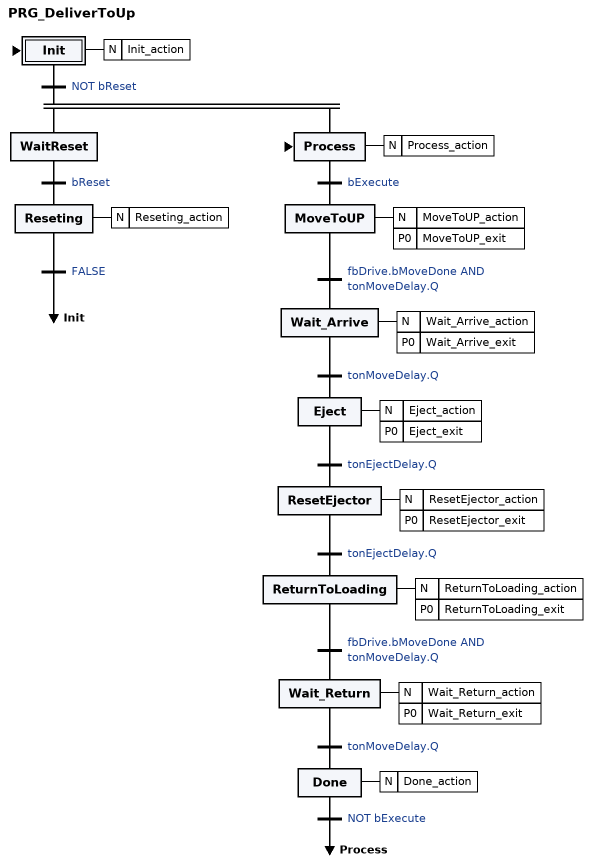
INITIAL_STEP Init:
	Init_action(N);
END_STEP
TRANSITION FROM Init TO (WaitReset, Process) := NOT bReset;
END_TRANSITION
STEP WaitReset:
END_STEP
TRANSITION FROM WaitReset TO Reseting := bReset;
END_TRANSITION
STEP Process:
	Process_action(N);
END_STEP
TRANSITION FROM Process TO MoveToUP := bExecute;
END_TRANSITION
STEP MoveToUP:
	MoveToUP_action(N);
	MoveToUP_exit(P0);
END_STEP
TRANSITION FROM MoveToUP TO Wait_Arrive := fbDrive.bMoveDone AND tonMoveDelay.Q;
END_TRANSITION
STEP Wait_Arrive:
	Wait_Arrive_action(N);
	Wait_Arrive_exit(P0);
END_STEP
TRANSITION FROM Wait_Arrive TO Eject := tonMoveDelay.Q;
END_TRANSITION
STEP Eject:
	Eject_action(N);
	Eject_exit(P0);
END_STEP
TRANSITION FROM Eject TO ResetEjector := tonEjectDelay.Q;
END_TRANSITION
STEP ResetEjector:
	ResetEjector_action(N);
	ResetEjector_exit(P0);
END_STEP
TRANSITION FROM ResetEjector TO ReturnToLoading := tonEjectDelay.Q;
END_TRANSITION
STEP ReturnToLoading:
	ReturnToLoading_action(N);
	ReturnToLoading_exit(P0);
END_STEP
TRANSITION FROM ReturnToLoading TO Wait_Return := fbDrive.bMoveDone AND tonMoveDelay.Q;
END_TRANSITION
STEP Wait_Return:
	Wait_Return_action(N);
	Wait_Return_exit(P0);
END_STEP
TRANSITION FROM Wait_Return TO Done := tonMoveDelay.Q;
END_TRANSITION
STEP Done:
	Done_action(N);
END_STEP
TRANSITION FROM Done TO Process := NOT bExecute;
END_TRANSITION
STEP Reseting:
	Reseting_action(N);
END_STEP
TRANSITION FROM Reseting TO Init := FALSE;
END_TRANSITION

ACTION Init_action:
SFCReset := FALSE;
bDone := FALSE;
END_ACTION

ACTION Process_action:
bDone := FALSE;
END_ACTION

ACTION MoveToUP_action:
bDone := FALSE;

fbDrive(
	bEnable:= TRUE,
	bStart:= TRUE,
	wTarget:= GPOS_PIPE_UP);

tonMoveDelay(IN:=TRUE , PT:= tMoveDelay);
END_ACTION

ACTION MoveToUP_exit:
fbDrive(
	bStart:= FALSE);

tonMoveDelay(IN:=FALSE);
END_ACTION

ACTION Wait_Arrive_action:
tonMoveDelay(IN:=TRUE , PT:= tMoveDelay);
END_ACTION

ACTION Wait_Arrive_exit:
tonMoveDelay(IN:=FALSE);
END_ACTION

ACTION Eject_action:
OEjector := TRUE;
tonEjectDelay(IN:=TRUE , PT:= tEjectorDelay);
END_ACTION

ACTION Eject_exit:
tonEjectDelay(IN:=FALSE);
END_ACTION

ACTION ResetEjector_action:
OEjector := FALSE;
tonEjectDelay(IN:=TRUE , PT:= tEjectorDelay);
END_ACTION

ACTION ResetEjector_exit:
tonEjectDelay(IN:=FALSE);
END_ACTION

ACTION ReturnToLoading_action:
fbDrive(
	bEnable:= TRUE,
	bStart:= TRUE,
	wTarget:= GPOS_LOADING);

tonMoveDelay(IN:=TRUE , PT:= tMoveDelay);
END_ACTION

ACTION ReturnToLoading_exit:
fbDrive(
	bStart:= FALSE);

tonMoveDelay(IN:=FALSE);
END_ACTION

ACTION Wait_Return_action:
tonMoveDelay(IN:=TRUE , PT:= tMoveDelay);
END_ACTION

ACTION Wait_Return_exit:
tonMoveDelay(IN:=FALSE);
END_ACTION

ACTION Done_action:
bDone := TRUE;
END_ACTION

ACTION Reseting_action:
SFCReset := TRUE;
END_ACTION
END_PROGRAM

(* POU OLD/PRG_DeliverToUp2, SFC *)
PROGRAM PRG_DeliverToUp2
VAR_INPUT
	bExecute: BOOL;
END_VAR
VAR_INPUT
	bDone: BOOL;
END_VAR
VAR
	tonMoveDelay	: TON;
	tonEjectDelay	: TON;
	tMoveDelay	: TIME := T#3s;
	tEjectorDelay	: TIME := T#3s;
END_VAR
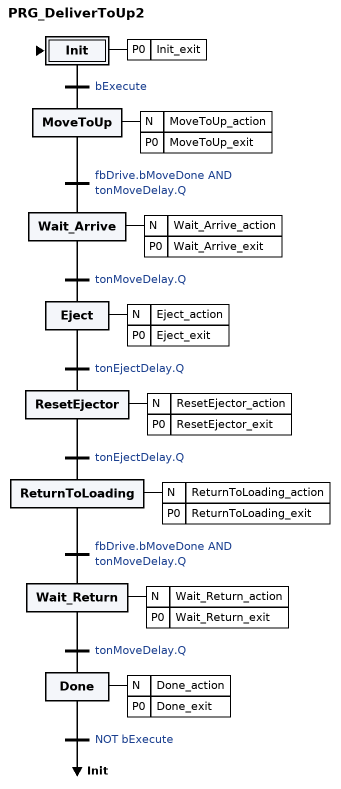
INITIAL_STEP Init:
	Init_exit(P0);
END_STEP
TRANSITION FROM Init TO MoveToUp := bExecute;
END_TRANSITION
STEP MoveToUp:
	MoveToUp_action(N);
	MoveToUp_exit(P0);
END_STEP
TRANSITION FROM MoveToUp TO Wait_Arrive := fbDrive.bMoveDone AND tonMoveDelay.Q;
END_TRANSITION
STEP Wait_Arrive:
	Wait_Arrive_action(N);
	Wait_Arrive_exit(P0);
END_STEP
TRANSITION FROM Wait_Arrive TO Eject := tonMoveDelay.Q;
END_TRANSITION
STEP Eject:
	Eject_action(N);
	Eject_exit(P0);
END_STEP
TRANSITION FROM Eject TO ResetEjector := tonEjectDelay.Q;
END_TRANSITION
STEP ResetEjector:
	ResetEjector_action(N);
	ResetEjector_exit(P0);
END_STEP
TRANSITION FROM ResetEjector TO ReturnToLoading := tonEjectDelay.Q;
END_TRANSITION
STEP ReturnToLoading:
	ReturnToLoading_action(N);
	ReturnToLoading_exit(P0);
END_STEP
TRANSITION FROM ReturnToLoading TO Wait_Return := fbDrive.bMoveDone AND tonMoveDelay.Q;
END_TRANSITION
STEP Wait_Return:
	Wait_Return_action(N);
	Wait_Return_exit(P0);
END_STEP
TRANSITION FROM Wait_Return TO Done := tonMoveDelay.Q;
END_TRANSITION
STEP Done:
	Done_action(N);
	Done_exit(P0);
END_STEP
TRANSITION FROM Done TO Init := NOT bExecute;
END_TRANSITION

ACTION Init_exit:
bDone := FALSE;
END_ACTION

ACTION MoveToUp_action:
fbDrive(
	bEnable:= TRUE,
	bStart:= TRUE,
	wTarget:= GPOS_PIPE_UP);

tonMoveDelay(IN:=TRUE , PT:= tMoveDelay);
END_ACTION

ACTION MoveToUp_exit:
fbDrive(
	bStart:= FALSE);
tonMoveDelay(IN:=FALSE);
END_ACTION

ACTION Wait_Arrive_action:
tonMoveDelay(IN:=TRUE , PT:= tMoveDelay);
END_ACTION

ACTION Wait_Arrive_exit:
tonMoveDelay(IN:=FALSE);
END_ACTION

ACTION Eject_action:
OEjector := TRUE;
tonEjectDelay(IN:=TRUE , PT:= tEjectorDelay);
END_ACTION

ACTION Eject_exit:
tonEjectDelay(IN:=FALSE);
END_ACTION

ACTION ResetEjector_action:
OEjector := FALSE;
tonEjectDelay(IN:=TRUE , PT:= tEjectorDelay);
END_ACTION

ACTION ResetEjector_exit:
tonEjectDelay(IN:=FALSE);
END_ACTION

ACTION ReturnToLoading_action:
fbDrive(
	bEnable:= TRUE,
	bStart:= TRUE,
	wTarget:= GPOS_LOADING);

tonMoveDelay(IN:=TRUE , PT:= tMoveDelay);
END_ACTION

ACTION ReturnToLoading_exit:
fbDrive(
	bStart:= FALSE);

tonMoveDelay(IN:=FALSE);
END_ACTION

ACTION Wait_Return_action:
tonMoveDelay(IN:=TRUE , PT:= tMoveDelay);
END_ACTION

ACTION Wait_Return_exit:
tonMoveDelay(IN:=FALSE);
END_ACTION

ACTION Done_action:
bDone := TRUE;
END_ACTION

ACTION Done_exit:
bDone := FALSE;
END_ACTION
END_PROGRAM

(* POU Programs/PRG_Sorting, SFC *)
PROGRAM PRG_Sorting
(*Template program for sorting operation*)
VAR_INPUT
	bReset		: BOOL := FALSE;	(*Reseting the SFC*)
	bExecute	: BOOL;			(*Executes PRG*)
END_VAR
VAR_OUTPUT
	bDone		: BOOL;		(*Program operations done*)
END_VAR
VAR
(* -------------INTERNAL-------------------*)
	bInitDone		: BOOL:=FALSE;	(*Initialisation done*)


(*System variables. See SFC-flags: http://infosys.beckhoff.com/content/1033/tcplccontrol/html/tcplcctrl_editorsfc.htm?id=24319#SFC-Flags*)
	SFCReset		: BOOL := FALSE;	(*For reseting the SFC*)
END_VAR
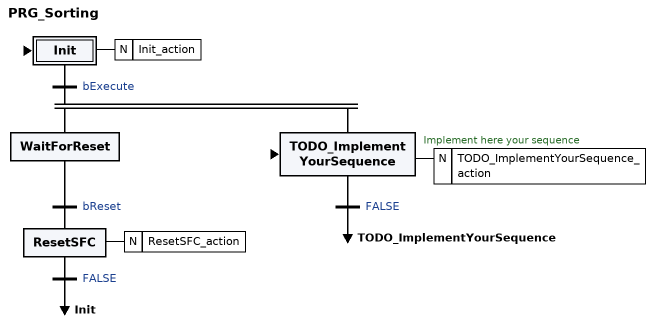
INITIAL_STEP Init:
	Init_action(N);
END_STEP
TRANSITION FROM Init TO (WaitForReset, TODO_ImplementYourSequence) := bExecute;
END_TRANSITION
STEP WaitForReset:
END_STEP
TRANSITION FROM WaitForReset TO ResetSFC := bReset;
END_TRANSITION
STEP TODO_ImplementYourSequence: (* Implement here your sequence *)
	TODO_ImplementYourSequence_action(N);
END_STEP
TRANSITION FROM TODO_ImplementYourSequence TO TODO_ImplementYourSequence := FALSE;
END_TRANSITION
STEP ResetSFC:
	ResetSFC_action(N);
END_STEP
TRANSITION FROM ResetSFC TO Init := FALSE;
END_TRANSITION

ACTION Init_action:
(*Clear Reset SFC*)
SFCReset:= FALSE;
END_ACTION

ACTION TODO_ImplementYourSequence_action:
(*Do some actions...

Sulje kaikki portit ... JA tarkista Steppiä seuraavassa transitioehdossa, että kaikki portit ovat kiinni
Close all gates.... and check in following transition that ALL gates are closed*)

;
END_ACTION

ACTION ResetSFC_action:
(*Reset SFC*)
SFCReset:=TRUE;
END_ACTION
END_PROGRAM

(* POU OLD/PRG_ToColourSensor, SFC *)
PROGRAM PRG_ToColourSensor
VAR_INPUT
	bReset		: BOOL;	(*Reset program*)
	bExecute		: BOOL;	(*enable and run*)
END_VAR
VAR_OUTPUT
	bDone			: BOOL;
END_VAR
VAR

	tonMoveDelay	: TON;
	SFCReset		: BOOL;
	tMoveDelay	: TIME := T#4s;
END_VAR
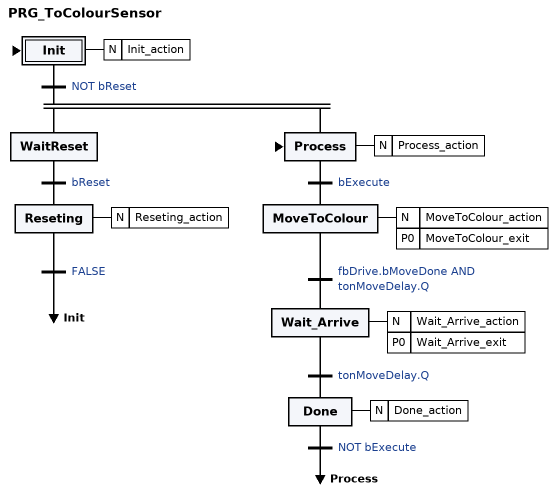
INITIAL_STEP Init:
	Init_action(N);
END_STEP
TRANSITION FROM Init TO (WaitReset, Process) := NOT bReset;
END_TRANSITION
STEP WaitReset:
END_STEP
TRANSITION FROM WaitReset TO Reseting := bReset;
END_TRANSITION
STEP Process:
	Process_action(N);
END_STEP
TRANSITION FROM Process TO MoveToColour := bExecute;
END_TRANSITION
STEP MoveToColour:
	MoveToColour_action(N);
	MoveToColour_exit(P0);
END_STEP
TRANSITION FROM MoveToColour TO Wait_Arrive := fbDrive.bMoveDone AND tonMoveDelay.Q;
END_TRANSITION
STEP Wait_Arrive:
	Wait_Arrive_action(N);
	Wait_Arrive_exit(P0);
END_STEP
TRANSITION FROM Wait_Arrive TO Done := tonMoveDelay.Q;
END_TRANSITION
STEP Done:
	Done_action(N);
END_STEP
TRANSITION FROM Done TO Process := NOT bExecute;
END_TRANSITION
STEP Reseting:
	Reseting_action(N);
END_STEP
TRANSITION FROM Reseting TO Init := FALSE;
END_TRANSITION

ACTION Init_action:
SFCReset := FALSE;
bDone := FALSE;
END_ACTION

ACTION Process_action:
bDone := FALSE;
END_ACTION

ACTION MoveToColour_action:
bDone := FALSE;

fbDrive(
	bEnable:= TRUE,
	bStart:= TRUE,
	wTarget:= GPOS_COLOR_SEN);

tonMoveDelay(IN:=TRUE , PT:= tMoveDelay);

(*
tonMoveDelay(IN:=TRUE , PT:= tMoveDelay);
*)
END_ACTION

ACTION MoveToColour_exit:
fbDrive(
	bStart:= FALSE);

tonMoveDelay(IN:=FALSE);
END_ACTION

ACTION Wait_Arrive_action:
tonMoveDelay(IN:=TRUE , PT:= tMoveDelay);
END_ACTION

ACTION Wait_Arrive_exit:
tonMoveDelay(IN:=FALSE);
END_ACTION

ACTION Done_action:
bDone := TRUE;
END_ACTION

ACTION Reseting_action:
SFCReset := TRUE;
END_ACTION
END_PROGRAM

(* POU OLD/PRG_ToColourSensor2, SFC *)
PROGRAM PRG_ToColourSensor2
VAR_INPUT
	bExecute: BOOL;
END_VAR
VAR_INPUT
	bDone: BOOL;
END_VAR
VAR
	tonMoveDelay	: TON;
	tonEjectDelay	: TON;
	tMoveDelay	: TIME := T#3s;
	tEjectorDelay	: TIME := T#3s;
END_VAR
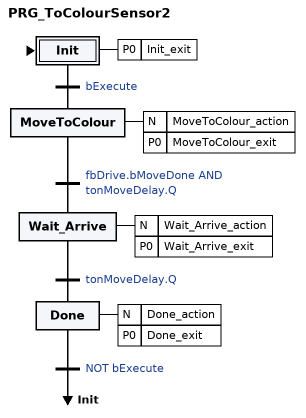
INITIAL_STEP Init:
	Init_exit(P0);
END_STEP
TRANSITION FROM Init TO MoveToColour := bExecute;
END_TRANSITION
STEP MoveToColour:
	MoveToColour_action(N);
	MoveToColour_exit(P0);
END_STEP
TRANSITION FROM MoveToColour TO Wait_Arrive := fbDrive.bMoveDone AND tonMoveDelay.Q;
END_TRANSITION
STEP Wait_Arrive:
	Wait_Arrive_action(N);
	Wait_Arrive_exit(P0);
END_STEP
TRANSITION FROM Wait_Arrive TO Done := tonMoveDelay.Q;
END_TRANSITION
STEP Done:
	Done_action(N);
	Done_exit(P0);
END_STEP
TRANSITION FROM Done TO Init := NOT bExecute;
END_TRANSITION

ACTION Init_exit:
bDone := FALSE;
END_ACTION

ACTION MoveToColour_action:
fbDrive(
	bEnable:= TRUE,
	bStart:= TRUE,
	wTarget:= GPOS_COLOR_SEN);

tonMoveDelay(IN:=TRUE , PT:= tMoveDelay);
END_ACTION

ACTION MoveToColour_exit:
fbDrive(
	bStart:= FALSE);
tonMoveDelay(IN:=FALSE);
END_ACTION

ACTION Wait_Arrive_action:
tonMoveDelay(IN:=TRUE , PT:= tMoveDelay);
END_ACTION

ACTION Wait_Arrive_exit:
tonMoveDelay(IN:=FALSE);
END_ACTION

ACTION Done_action:
bDone := TRUE;
END_ACTION

ACTION Done_exit:
bDone := FALSE;
END_ACTION
END_PROGRAM

(* POU FBs/FB_StateModel_ST, ST *)
FUNCTION_BLOCK FB_StateModel_ST
(*PackML State model implementation. Slightly modified implementation.
Author: 	Niko Siltala, niko.siltala@tut.fi
Date: 	2016-01-29
*)
VAR_INPUT
	bResetFB	: BOOL;		(*Resets whole FB*)
	eModeReq	: E_ModeCtrl;	(*Requested mode*)
	wIgnoreState	: DWORD;	(*Ignoring states. See bit from E_State definition. Aborting = bit0*)
	bSC			: BOOL;		(*Step Completed acknoledgement*)
	bAbort		: BOOL;		(*Abortting signal = EmergencyStop*)
	bClear		: BOOL;		(*Clear signal*)
	bReset		: BOOL;		(*Reseting signal*)
	bStart		: BOOL;		(*Start signal*)
	bHold		: BOOL;		(*Hold signal*)
	bUn_Hold	: BOOL;		(*Un-Hold signal*)
	bSuspend	: BOOL;		(*Suspend signal*)
	bUn_Suspend	: BOOL;		(*Un-Suspend signal*)
	bStop		: BOOL;		(*Stop signal*)
	bComplete	: BOOL;		(*Complete signal*)
	bAck_Completed	: BOOL;	(*Acknoledgement for Complete signal*)
END_VAR
VAR_OUTPUT
	eMode	: E_ModeCtrl;	(*Current mode*)
	eState	: E_State;	(*Current state*)
END_VAR
VAR
	RTrig_bSC	: R_TRIG; 	(*Rising trigger for State Completed*)
	RTrig_StateChange	: R_TRIG; 	(*Rising trigger for State signal*)
	bResetLocal		: BOOL:=FALSE;	(*Paikallinen Reset*)
	bInitDone	: BOOL;		(*Initialisation*)
END_VAR
IF bResetFB THEN	(*Reseting FB*)
	bInitDone := FALSE;
END_IF;

(*Initialisation*)
IF NOT bInitDone THEN
	eState:= eSt_Aborting;
	bInitDone:=TRUE;
END_IF;

(*Rising triggers monitor*)
RTrig_bSC(CLK:=bSC , Q=> );

(*Abort signal interrupt*)
IF bAbort AND (eState > eSt_Clearing) THEN
	eState:=eSt_Aborting;
END_IF;

(*Stop signal interrupt*)
IF bStop AND (eState > eSt_Stopping) THEN
	eState:=eSt_Stopping;
END_IF;


(*Main case structure*)
CASE eState OF
eSt_Aborting:
	IF bSC THEN
		eState:=eSt_Aborted;
	END_IF;

eSt_Aborted:
	eMode:=eModeReq;	(*Change Mode*)
	IF bClear AND NOT bAbort THEN
		eState:=eSt_Clearing;
	END_IF;

eSt_Clearing:
	IF bAbort THEN
		eState:=eSt_Aborting;
	ELSIF bSC THEN
		eState:=eSt_Stopped;
		RTrig_StateChange(CLK:=bReset , Q=> );
	END_IF;

eSt_Stopping:
	IF bSC THEN
		eState:=eSt_Stopped;
		RTrig_StateChange(CLK:=bReset , Q=> );
	END_IF;

eSt_Stopped:
	eMode:=eModeReq;	(*Change Mode*)
	RTrig_StateChange(CLK:=bReset , Q=> );
(*	ELSIF NOT bStop AND (RTrig_StateChange.Q OR (wIgnoreState.5 AND bStart) ) THEN*)
	IF NOT bStop THEN	(*Stop signal is not active.*)
		IF wIgnoreState.5 AND bStart THEN	(*Reset state is ignored and going directly to start *)
			eState:=eSt_Idle;
		ELSIF RTrig_StateChange.Q THEN 	(*Rising edge for reset*)
			eState:=eSt_Resetting;
		END_IF;
	END_IF;

eSt_Resetting:
	IF bSC OR wIgnoreState.5 THEN
		eState:=eSt_Idle;
	END_IF;

eSt_Idle:
	eMode:=eModeReq;	(*Change Mode*)
	IF bStart OR wIgnoreState.6 THEN
		eState:=eSt_Starting;
	END_IF;

eSt_Starting:
	IF bSC OR wIgnoreState.7 THEN
		eState:=eSt_Execute;
	END_IF;

eSt_Execute:
	IF bComplete THEN
		eState:=eSt_Completing;
	ELSIF bHold THEN
		eState:=eSt_Holding;
	ELSIF bSuspend THEN
		eState:=eSt_Suspending;
	END_IF;

eSt_Holding:
	IF bSC THEN
		eState:=eSt_Held;
	END_IF;

eSt_Held:
	IF bUn_Hold AND NOT bHold THEN
		eState:=eSt_UnHolding;
	END_IF;

eSt_UnHolding:
	IF bSC THEN
		eState:=eSt_Execute;
	END_IF;

eSt_Suspending:
	IF bSC THEN
		eState:=eSt_Suspended;
	END_IF;

eSt_Suspended:
	IF bUn_Suspend AND NOT bSuspend THEN
		eState:=eSt_Unsuspending;
	END_IF;

eSt_Unsuspending:
	IF bSC THEN
		eState:=eSt_Execute;
	END_IF;

eSt_Completing:
	IF RTrig_bSC.Q THEN
		eState:=eSt_Completed;
	END_IF;

eSt_Completed:
	IF bAck_Completed THEN
		eState:=eSt_Resetting;
	END_IF;

ELSE
	(*Default error handler. Undefined state set*)
	eState:=eSt_Aborting;
END_CASE;
END_FUNCTION_BLOCK

(* POU OLD/FB_TransferBall, ST *)
FUNCTION_BLOCK FB_TransferBall
VAR_INPUT
	bExecute			: BOOL;	(*enable and run*)
	bBallToTransfer 	: E_BallColour;
END_VAR
VAR_OUTPUT
	bDone			: BOOL;
	bActDone		: BOOL := FALSE;
END_VAR
VAR
	tonMoveDelay	: TON;
	tonEjectDelay	: TON;
	tMoveDelay	: TIME := T#1s;
	tEjectorDelay	: TIME := T#1s;
END_VAR
IF bExecute THEN
	CASE bBallToTransfer OF
		Yellow:
			PRG_DeliverToUp2( bExecute:= TRUE , bDone=> );
				bDone	:= FALSE;
				IF PRG_DeliverToUp2.bDone THEN
					PRG_DeliverToUp2(bExecute:=FALSE);
					bDone	:= TRUE;
				END_IF
		Blue:
			PRG_DeliverToMid2( bExecute:= TRUE, bDone=> );
				bDone	:= FALSE;
				IF PRG_DeliverToMid2.bDone THEN
					PRG_DeliverToMid2(bExecute:=FALSE);
					bDone	:= TRUE;
				END_IF
		Red, NoColour:
			PRG_DeliverToGarbage2( bExecute:= TRUE, bDone=> );
				bDone	:= FALSE;
				IF PRG_DeliverToGarbage2.bDone THEN
					PRG_DeliverToGarbage2( bExecute:=FALSE);
					bDone	:= TRUE;
				END_IF
	ELSE
		PRG_DeliverToMid2(bExecute:=FALSE);
		PRG_DeliverToUp2(bExecute:=FALSE);
		PRG_DeliverToGarbage2( bExecute:=FALSE);
		bDone	:= FALSE;
	END_CASE
ELSE
	bDone := FALSE;
END_IF
END_FUNCTION_BLOCK

(* Visualisation FBs_Visu/FB_DriveMovement2
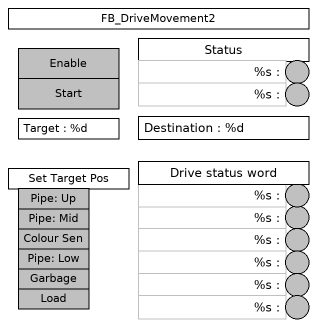
rectangle at (0,0)-(301,21): text "FB_DriveMovement2"
embedded screen at (130,30)-(301,311): FB_VC_Drive_Status
rectangle at (10,110)-(111,131): text "Target : %d"; shows $FB$.wTarget
rectangle at (10,40)-(111,71): text "Enable"; alarm colour if $FB$.bEnable; toggles $FB$.bEnable
rectangle at (10,70)-(111,101): text "Start"; alarm colour if $FB$.bStart; toggles $FB$.bStart
rectangle at (10,280)-(81,301): text "Load"; alarm colour if $FB$.wTarget = .GPOS_LOADING; runs INTERN ASSIGN $FB$.wTarget:=(GPOS_LOADING)
rectangle at (10,260)-(81,281): text "Garbage"; alarm colour if $FB$.wTarget = .GPOS_GARBAGE; runs INTERN ASSIGN $FB$.wTarget:=(GPOS_GARBAGE)
rectangle at (0,160)-(121,181): text "Set Target Pos"
rectangle at (10,240)-(81,261): text "Pipe: Low"; alarm colour if $FB$.wTarget = .GPOS_PIPE_LOW; runs INTERN ASSIGN $FB$.wTarget:=(GPOS_PIPE_LOW)
rectangle at (10,220)-(81,241): text "Colour Sen"; alarm colour if $FB$.wTarget = .GPOS_COLOR_SEN; runs INTERN ASSIGN $FB$.wTarget:=(GPOS_COLOR_SEN)
rectangle at (10,200)-(81,221): text "Pipe: Mid"; alarm colour if $FB$.wTarget = .GPOS_PIPE_MID; runs INTERN ASSIGN $FB$.wTarget:=(GPOS_PIPE_MID)
rectangle at (10,180)-(81,201): text "Pipe: Up"; alarm colour if $FB$.wTarget = .GPOS_PIPE_UP; runs INTERN ASSIGN $FB$.wTarget:=(GPOS_PIPE_UP)
1 more shapes without text or variables
*)

(* Visualisation FBs_Visu/FB_VC_Drive_Status
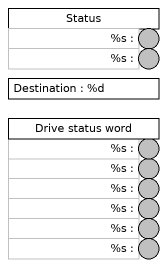
embedded screen at (0,150)-(151,171): VC_BOOLEANSTATUS
rectangle at (0,0)-(151,21): text "Status"
embedded screen at (0,170)-(151,191): VC_BOOLEANSTATUS
embedded screen at (0,130)-(151,151): VC_BOOLEANSTATUS
embedded screen at (0,190)-(151,211): VC_BOOLEANSTATUS
embedded screen at (0,210)-(151,231): VC_BOOLEANSTATUS
embedded screen at (0,230)-(151,251): VC_BOOLEANSTATUS
rectangle at (0,70)-(151,91): text "Destination : %d"; shows $FB$.wDestination
rectangle at (0,110)-(151,131): text "Drive status word"
embedded screen at (0,20)-(151,41): VC_BOOLEANSTATUS
embedded screen at (0,40)-(151,61): VC_BOOLEANSTATUS
*)

(* Visualisation V_DRIVE
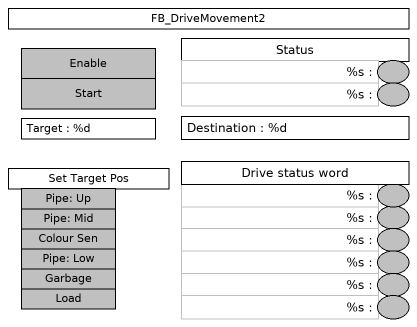
embedded screen at (0,0)-(401,311): FB_DriveMovement2
*)

(* Visualisation V_MAIN
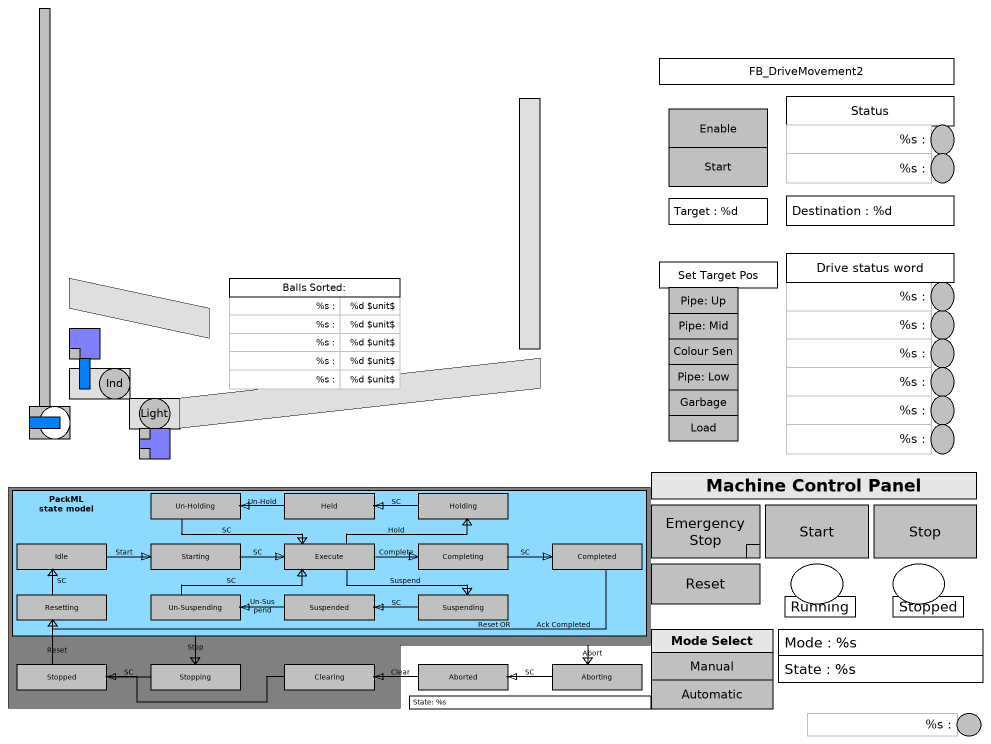
embedded screen at (60,320)-(531,451): VC_Graph_Sorter
embedded screen at (20,0)-(61,431): VC_Graph_Lift
embedded screen at (220,270)-(391,381): VC_Graph_Counters
embedded screen at (-1,479)-(642,701): VC_PackMLStates
embedded screen at (642,464)-(974,701): VC_Panel_MachineControl
embedded screen at (650,50)-(945,446): FB_DriveMovement2
embedded screen at (798,705)-(972,728): VC_BOOLEANSTATUS
2 more shapes without text or variables
*)

(* Visualisation Components/VC_BOOLEANSTATUS
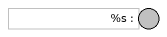
rectangle at (0,0)-(131,21): text "%s :"; shows $Name$
ellipse at (130,0)-(151,21): alarm colour if $bFlag$
*)

(* Visualisation Components/VC_Graph_Counters
